Staubli VAL3: user.pjx

--- user.pjx ---
Parameters version=s7.4 stackSize=5000 millimeterUnit=true
Program file=start.pgx
Program file=stop.pgx
Data file=user.dtx

--- userPage7En.dtx ---
public num nBottomX[2]
  [0] = 21
  [1] = 21
public num nBottomY = 10
num nFirst
num nKey = 255
num nOldValue[2]
  [0] = 200
  [1] = 200
public num nPage = 100000
public num nTopX[2]
  [0] = 17
  [1] = 17
public num nTopY
public num nView
string sExample1
string sExample2
public string sItems[17]
  [0] = "Name: > "
  [1] = "coord  X > 680.52"
  [2] = "coord  Y > -61.92"
  [3] = "coord  Z > 300.32"
  [4] = "coord RX > -10   "
  [5] = "coord RY > 175.5 "
  [6] = "coord RZ > 68.47"
  [7] = "Axis pos > 90   "
  [8] = "MoveType > Linear"
  [9] = "Speed    > 600 mm/s"
  [10] = "Accelerat> 200 %"
  [11] = "Stop  > [ ]"
  [12] = "Blend[x] > 30 mm"
  [13] = "Action : 1> "
  [14] = "Action : 2> "
  [15] = "Action : 3> "
  [16] = "Anticipation > 0 mm"
string sMenu
string sMessage[3]
  [0] = "Insert the speed, all the points that"
  [1] = "have the same speeed will be change,"
  [2] = "use mm/sec >600"
string sTab[4]
  [0] = "test1"
  [1] = "test2"
  [2] = "test3"
  [3] = "test4"
string sTitle
bool Show
bool bReadWrite[17]
  [0] = true
  [1] = true
  [2] = true
  [3] = true
  [4] = true
  [5] = true
  [6] = true
  [7] = true
  [8] = true
  [9] = true
  [10] = true
  [11] = true
  [12] = true
  [13] = true
  [14] = true
  [15] = true
  [16] = true
public bool bShowDialog
public bool bUseEscape = true
public bool bUseRefresh
screen scr

--- start.pgx ---
program start()
begin
  call example1()
end

--- changeValue.pgx ---
public program changeValue(screen& x_scr, num& x_nValue[], num x_nMin, num x_nMax, num x_nX, num x_nY, string& x_sItem[])
  local num l_nOldValue[2]
  local string l_sItem
  local string l_sMessage
  local string l_sEmpty
  local bool l_bComma
begin
  //-----------------------------------------------------------------------
  //Header begin 开头
  //Description of program  程序的描述
  //  Get a numerical value on the x_nX column and x_nY line and test if    在x_nX列和x_nY行得到一个数值量，测试
  //  the value is between x_nMin and x_nMax. If the two parameters x_nMin  这个值是否在x_nMin和x_nMax之间。如果这两个参数x_nMin
  //  and x_nMax are equal there are no limits.                             和x_nMax值相等的，那这里就没有限制了。
  //  If x_sItems is not Empty, the program displays the list of Items and  如果x_sItems是非空的，程序显示了条目的列表
  //  you can change the selected Item : the index is returned in x_nValue. 你可以改变已选的条目：索引回到了x_nValue
  //
  //Input parameters  输入参数
  //  num x_nMin :    x_nMin的数值：
  //    role : min value limit  作用：最小值的限制
  //  num x_nMax :    x_nMax的数值：
  //    role : max value limit  作用：最大值的限制
  //  num x_nX :      x_nX的数值：
  //    role : X cursor position for change the value  作用：X光标的位置变化值
  //  num x_nY :      x_nY的数值
  //    role : Y cursor position for change the value  作用：Y光标的位置变化值
  //
  //Output paramaters  输出参数
  //  num x_nValue :   x_nValue的数值
  //    role : numerical value changed or index pointer of x_sItem  作用：x_sItem的数值量改变或者索引指针
  //  string x_sItems  x_sItems的字符串
  //    role : array of Items  作用：条目的数组
  //
  //Example 例子
  //  call changeValue(scrMy,l_nValue,0,10,2,5,"") //The user can changed the numerical  用户可以改变l_nValue的数值量
  //                                           value of l_nValue. If the seized          如果得到的值不在0到10范围内，
  //                                           is not between 0 to 10 the user must      用户必须改变这个值。
  //                                           changed the value.
  //
  //  call changeValue(scrMy,l_nValue,0,10,2,5,sItem) //The list sItem is displaying on  列表条目是正在显示在屏幕上，
  //                                              the screen and the user select one     用户可以选择列表中的某个元素。
  //                                              element of the list. The index         索引会回到l_nValue中。
  //                                              is returned in l_nValue.
  //
  //
  //History  历史
  //  Creation : 28-04-08 - f.Rob  创建：28-04-08 - f.Rob
  //  Modified : 08-08-11 - J.Cook 修改：08-08-11 - J.Cook
  //                                   Changed $setTextMode to setTextMode  改变$setTextMode到setTextMode
  //                                   And replaced literals ("", 0) with local variables
  //                                   when passing parameters by reference
  //
  //  Modified : 08-08-22 - J.Cook     Add screen parameter 增加屏幕参数
  //Header end  结束
  //-----------------------------------------------------------------------
  //
  if x_nMin>x_nMax
    return
  endIf
  //Print the line in white  已白色打印该行
  call nullKey(x_scr,nKey)
  l_nOldValue[1]=round(x_nValue)
  x_nValue=(round(x_nValue*100))/100
  l_nOldValue=x_nValue
  //Check if is using the comma or not  检查有没有使用逗号
  if l_nOldValue!=l_nOldValue[1]
    l_bComma=true
  else
    l_bComma=false
  endIf
  //Start  开始
  call clear(x_scr, 0,13)
  do
    if x_sItem==""
      //Use the get num  使用得到数值
      if l_bComma
        call strFill(l_sEmpty,len(toString(".2",x_nValue)),l_sEmpty)
      else
        call strFill(l_sEmpty,len(toString("",x_nValue)),l_sEmpty)
      endIf
      call type(x_scr, x_nX,x_nY,l_sEmpty)
      gotoxy(x_scr, x_nX,x_nY)
      nKey=get(x_scr, x_nValue)
      // CHECK for MIN MAX VALUE 检查最大最小值
      if x_nMax!=x_nMin
        if x_nValue>x_nMax
          //Ask if you want to continue  询问是否你想要继续
          popUpMsg("MAX: "+toString(".2",x_nMax))
          x_nValue=l_nOldValue
          //x_nValue=x_nMax
          nKey=-1
        else
          if x_nValue<x_nMin
            popUpMsg("MIN: "+toString(".2",x_nMin))
            //x_nValue=x_nMin
            x_nValue=l_nOldValue
            nKey=-1
          endIf
        endIf
      endIf
      // UPDATE THE VALUE 更新数值
      if l_bComma
        call type(x_scr, x_nX,x_nY,toString(".2",x_nValue))
      else
        call type(x_scr, x_nX,x_nY,toString("",x_nValue))
      endIf
    else
      // STRING CHOICE 字符串选择
      nKey=getKey(x_scr)
      switch nKey
        // CHANGE THE ITEMS ARRAY  改变条目数组
        case 261
          // UP
          x_nValue=abs((x_nValue+1)%size(x_sItem))
        break
        case 266
          // DOWN
          x_nValue=abs((x_nValue+size(x_sItem)-1)%size(x_sItem))
        break
      endSwitch
      // UPDATE THE VALUE 更新数值
      setTextMode(x_scr, 3)
      call typeLen(x_scr,x_nX,x_nY,x_sItem[x_nValue],10)
      setTextMode(x_scr, 0)
    endIf
    //Release the resource  释放资源
    delay(0)
  until nKey==270 or nKey==255
  if nKey==255
    bUseEscape=true
    x_nValue=l_nOldValue
    if x_sItem!=""
      x_sItem=x_sItem[l_nOldValue]
    endIf
  else
    bUseEscape=false
  endIf
  //Leave the resource  离开资源
  delay(0)
end

--- clear.pgx ---
public program clear(screen& x_scr, num x_nX, num x_nY)
  local num i
  local num lLen
begin
  //-----------------------------------------------------------------------
  //Header begin 开头
  //Description of program  程序描述
  //  Erase the pY line from the column pX of the userPage.
  //  在用户界面中，擦除pX列中的PY行
  //Input parameters  输入参数
  //  num x_nX :
  //    role : Cursor column  作用：光标列
  //    possible value : 0 to 39  可能的值：0到39
  //  num x_nY :
  //    role : Cursor row     作用：光标行
  //    possible value : 0 to 13  可能的值：0到39
  //
  //Example 例子
  //  call clear(scrMy,15,8)
  //
  //History  历史
  //  Creation : 28-04-08 - f.Rob
  //
  //  Modified : 22 Aug 2011 - J. Cook  Added user screens
  //Header end 结束
  //-----------------------------------------------------------------------
  call typeLen(x_scr, x_nX,x_nY," ",40-x_nX)
  gotoxy(x_scr, x_nX,x_nY)
end

--- divideString.pgx ---
program divideString(string& x_sMsg[], num& x_nLine[])
  local string l_sCopyMsg
  local num l_nLength
  local string l_sSwap
  local num l_nFlag
  local num l_nTotalFlag
  local string l_sCR
  local num l_nPosCR
begin
  //-----------------------------------------------------------------------
  //Header begin 开头
  //Description of program  程序描述
  //  Divide a message if it is too long.  如果它够长的话，划分一条消息
  //  The program search a space for cut the message. 程序去搜寻一个空间为的是分割消息
  //  Return the numbers of lines used for writing the message.
  //
  //Input parameters  输入参数
  //  string x_sMsg : 字符串x_sMsg
  //    role : Message that you want to display  作用：你想去展示的消息
  //  num x_sLine :   数值量x_sLine
  //    role : Numbers of the lines that will be use  作用：该行的数值将会被使用
  //
  //Example  例子
  //  call divideString("Staubli Robotics : example userPage library",l_nLine)
  //
  //History
  //  Creation : 28-04-08 - f.Rob
  //Header end 结束
  //-----------------------------------------------------------------------
  //Carriage return  回车
  l_sCR="#"
  x_nLine=0
  //Length of a line for a message 一条消息一行的长度
  l_nLength=38
  //Copy the message  复制该信息
  l_sCopyMsg=x_sMsg
  //First case  第一种情况
  call findPos(l_sCopyMsg,l_sCR,l_nPosCR)
  if (getDisplayLen(l_sCopyMsg)>l_nLength-1) or (l_nPosCR!=-1)
    //Compose the message  重组这条消息
    do
      l_sSwap=l_sCopyMsg
      //Set the x_sMsg
      if size(x_sMsg)-1<x_nLine
        insert(x_sMsg[x_nLine])
      endIf
      call findPos(l_sCopyMsg,l_sCR,l_nPosCR)
      if (getDisplayLen(l_sCopyMsg)>l_nLength-1 or (l_nPosCR!=-1)) and x_nLine<8
        //Divide the string 分割字符串
        l_nTotalFlag=0
        call findPos(l_sCopyMsg,l_sCR,l_nPosCR)
        //Divide the string
        if l_nPosCR!=-1 and l_nPosCR<l_nLength
          //Carriage return  回车
          call leftPos(l_sCopyMsg,l_nPosCR,l_sSwap)
          //l_sSwap=left(l_sCopyMsg,l_nPosCR)
          call rightPos(l_sCopyMsg,getDisplayLen(l_sCopyMsg)-(l_nPosCR)-1,l_sCopyMsg)
          //l_sCopyMsg=right(l_sCopyMsg,len(l_sCopyMsg)-(l_nPosCR)-1)
          if getDisplayLen(l_sSwap)==0
            l_sSwap=" "
          endIf
        else
          //Search for the space then return 搜索空间然后返回
          do
            call findPos(l_sSwap," ",l_nFlag)
            //l_nFlag=find(l_sSwap," ")
            if l_nFlag!=-1 and l_nFlag<=l_nLength
              //l_sSwap=right(l_sSwap,len(l_sSwap)-l_nFlag-1)
              call rightPos(l_sSwap,getDisplayLen(l_sSwap)-l_nFlag-1,l_sSwap)
              l_nTotalFlag=l_nTotalFlag+l_nFlag+1
            else
              if l_nTotalFlag==0 and (l_nFlag==-1 or l_nFlag>l_nLength)
                l_nFlag=-1
                l_nTotalFlag=38
              endIf
            endIf
          until l_nTotalFlag>=l_nLength+2 or l_nFlag==-1
          //Normal
          if l_nTotalFlag==0
            //Full line  整行
            call leftPos(l_sCopyMsg,l_nLength,l_sSwap)
            //l_sSwap=left(l_sCopyMsg,l_nLength)
            //l_sCopyMsg=right(l_sCopyMsg,len(l_sCopyMsg)-l_nLength)
            call rightPos(l_sCopyMsg,getDisplayLen(l_sCopyMsg)-l_nLength,l_sCopyMsg)
          else
            //Divide it
            call leftPos(l_sCopyMsg,l_nTotalFlag-l_nFlag-2,l_sSwap)
            //l_sSwap=left(l_sCopyMsg,l_nTotalFlag-l_nFlag-2)
            //l_sCopyMsg=right(l_sCopyMsg,len(l_sCopyMsg)-(l_nTotalFlag-l_nFlag-1))
            call rightPos(l_sCopyMsg,getDisplayLen(l_sCopyMsg)-(l_nTotalFlag-l_nFlag-1),l_sCopyMsg)
          endIf
        endIf
        //Set the string  设置字符串
        x_sMsg[x_nLine]=l_sSwap
        x_nLine=x_nLine+1
      else
        //Limit the string  限制字符串
        call rightPos(l_sSwap,l_nLength,x_sMsg[x_nLine])
        //x_sMsg[x_nLine]=right(l_sSwap,l_nLength)
        l_sSwap=""
      endIf
    until l_sSwap==""
  endIf
end

--- editNumField.pgx ---
public program editNumField(screen& x_scr, string x_sTitle, string& x_sItemName[], num& x_nItem[], num& x_nMin[], num& x_nMax[])
  local num j
  local num l_nSize
  local num l_nKey
  local string l_sEvent
  local num l_nIndex
  local num l_nField
  local string l_sItem
  local string l_sEmpty
begin
  //-----------------------------------------------------------------------
  //Header begin 开头
  //Description of program  程序描述
  //  Modify numerical values of a list of Items. 修改条目列表的数值量
  //  When you use this program it creates automatically the list of x_sItemName. 当你使用这个程序，它能够自动创建x_sItemName的列表
  //  You can navigate and select the Item that you want to modify the value.     你能够导航和选择你想修改值的条目
  //  If you press on ESC you quit this list and all values that you have entered 如果你按压ESC键，你会退出这个列表，你已经输入的所有值
  //  will not be saved.                                                          将不会被保存
  //  You can use an array for the parameters min and max to add limits           你能够使用一个针对最小值最大值的参数的数组去增加
  //  for every Items.                                                            每一个条目的限制
  //  If the parameters min and max are equal there are no limits.                如果参数的最小值和最大值是相等的，那儿就没有限制。
  //
  //Input parameters  输入参数：
  //  string x_sTitle :  字符串x_sTitle
  //    role : Title of the list  作用：列表的标题
  //
  //Output parameters  输出参数
  //  string x_sItemName : 字符串x_sItemName：
  //    role : array of Items that you want to edit the numerical values 作用：你想要编辑的条目数组的数值量
  //  num x_nItem :  数值量x_nItem
  //    role : array of values corresponding of the Items  作用：对应条目的数组值
  //  num x_nMin :  数值量x_nMin
  //    role : minimum limit for x_nItem values  作用：x_nItem值的最小值限制
  //  num x_nMax    数值量x_nMax
  //    role : maximum limit for x_nItem values  作用：x_nItem值的最大值限制
  //
  //Example 例子
  //  call editNumField(scrMy,"Menu",sItem,nItem,nMin,nMax)
  //
  //History
  //  Creation : 28-04-08 - f.Rob
  //  Modified : 08-08-11 - J.Cook     Changed $setTextMode to setTextMode
  //                                   And replaced literals ("", 0) with local variables
  //                                   when passing parameters by reference
  //
  //  Modified : 08-08-22 - J.Cook     Add screen parameter
  //Header end 结束
  //-----------------------------------------------------------------------
  l_sEmpty = ""
  nView=nFirst=0
  //Copy all the values x_nItem 复制所有的x_nItem的值
  call numCopy(x_nItem,nOldValue)
  l_nSize=size(x_nItem)-1
  //Create the LIST  创建列表
  call setSizeList(7,max((6-l_nSize/2)-2,2),23,min((l_nSize+1),8))
  call listCreate(x_scr, x_sTitle)
  //Insert Items  插入条目
  for j=0 to l_nSize
    l_sItem=x_sItemName[j]
    call strlength(l_sItem,15)
    call listAdd(l_sItem+": "+toString(".1",x_nItem[j]))
  endFor
  call listUpdate(x_scr, 0)
  do
    call clear(x_scr, 0,13)
    call typeMenu(x_scr, 8,"OK")
    l_nKey=get(x_scr)
    call listEvent(x_scr, l_nKey,l_nIndex,l_sEvent)
    //On Enter Key  在回车键
    if l_nKey==270
      call listCursor(x_scr,nView,false)
      if size(x_nMin)==size(x_nItem)
        //Use min and max  使用最小值和最大值
        call changeValue(x_scr, x_nItem[l_nIndex],x_nMin[l_nIndex],x_nMax[l_nIndex],15+10,nView+nTopY+1,l_sEmpty)
      else
        call changeValue(x_scr,x_nItem[l_nIndex],0,0,15+10,nView+nTopY+1,l_sEmpty)
      endIf
      //UPDATE 更新
      call listDel(l_nIndex)
      l_sItem=x_sItemName[l_nIndex]
      call strlength(l_sItem,15)
      call listIns(l_sItem+": "+toString(".1",x_nItem[l_nIndex]),l_nIndex)
      call listUpdate(x_scr,l_nIndex-nView)
    endIf
    delay(0)
  until l_nKey==278 or l_nKey==255
  //Escape use????
  if l_nKey==255
    bUseEscape=true
    call numCopy(nOldValue,x_nItem)
  else
    bUseEscape=false
  endIf
  //Exit
  call nullKey(x_scr,l_nKey)
end

--- example.pgx ---
program example()
  local num l_nKey
  local num l_nItem[2]
  local num l_nView[2]
  local string l_sItem
  local string l_sMsg
  local string l_sButton[2]
  local num i
  local bool l_bLarge
  local bool l_bQuit
  local string l_sMenu
  local num l_nSeconds
  local string l_sHourMinSec
  local string l_sItemName[5]
  local num l_nItemExample[5]
  local num l_nMaxExample[5]
  local num l_nMinExample[5]
  local num l_nMenu
  local num l_nSelected[2]
  local bool l_bExit
  local num l_nFirst[2]
  local string l_sEmpty
  local string l_sText
  local num l_nZero
begin
  //-----------------------------------------------------------------------
  //Header begin 开头
  //Description of program 程序的描述
  //  This is an example for use this library. 这是一个使用库的例子程序。
  //  This example performs the following actions : 该程序执行以下动作：
  //  - Run the fhmns program (converted of num seconds in string hour) 运行fhmns程序(时间转换程序，把秒数转换成几时几分几秒的形式)
  //  - add, insert, delete, and select an Item with an updating of the menu. 用一个更新的菜单显示增加，插入，删除和选择一个条目
  //  - change Menu (list of Items) with left and right keys 用左右键改变菜单（条目列表）
  //  - clear the menu  清除菜单
  //  - Run a simple list (no array) for just test the scrolling 运行一个简单的列表（没有数组），只为了测试列表滚动条
  //
  //  The sequence is : 这个顺序是：
  //  - Creation of 2 string arrays for the lists of items 条目列表里创建两个字符串数组
  //  - Start main loop 开始主循环
  //  -   Creation of the menu with 2 lists  2个列表菜单的创建
  //  -   Reading events from the keyboard   从键盘中读取事件
  //  -     case TAB           : update the width of the list (enlarge/reduce)  TAB键：更新列表的宽度（扩大/减少）
  //  -     case left or right : update the item's list and change the menu    左右键：更新条目的列表和改变菜单
  //  -     case Enter         : displays the Item selected                    回车键：显示已选的条目
  //  -     case F1 or ESC     : quit the program                           F1或ESC键：退出程序
  //  -     case F2            : clear th list                                   F2键：清除列表
  //  -     case F3            : Run function wich converted seconds             F3键：运行时间转换函数
  //                              -> string Hours:Min:Sec                              由s转换成h：m：s的形式
  //  -     case F4            : test editNumField() function                    F4键：测试editNumField()函数
  //  -     case F5            : creation of an other list : simple list         F5键：创建一个其他列表：简单列表
  //  -     case F6            : delete an Item                                  F6键：删除一个条目
  //  -     case F7            : add an item at the end of the list              F7键：在列表末端增加一个条目
  //  -     case F8            : insert an item at the current position          F8键：在当前的位置插入一个条目
  //  -   Update the Item's list                                                 更新条目的列表
  //  -   Refresh the screen                                                     刷新屏幕
  //
  //History                                                                      历史
  //  Creation : 28-04-08 - f.Rob                                                创建：28-04-08 - f.Rob
  //  Modified : 08-08-11 - J.Cook     Changed $setTextMode to setTextMode       修改：08-08-11 - J.Cook
  //                                   And replaced literals ("", 0) with local variables
  //                                   when passing parameters by reference
  //Header end  结束
  //-----------------------------------------------------------------------
  l_sEmpty = ""
  cls(scr)
  userPage(scr)
  //---------------------------------------------------
  // CREATION OF 2 STRING ARRAYS FOR THE LISTS OF ITEMS 为这个项目的列表创建2字符串数组
  //---------------------------------------------------
  //Empty the two lists  清空这两个列表
  call stringCopy(l_sEmpty,sExample1)
  call stringCopy(l_sEmpty,sExample2)
  //Build the first list  建立第一个列表
  for i=0 to 19
    if sExample1!=""
      append(sExample1)
    endIf
    sExample1[i]="Program "+toString("",i)
  endFor
  //Build the second list  建立第二个列表
  for i=0 to 14
    if sExample2!=""
      append(sExample2)
    endIf
    sExample2[i]="Item "+toString("",i)
  endFor
  //----------------
  // START THE LOOP   开始循环
  //----------------
  do
    //-------------------------------------
    // CREATION OF THE MENU WITH TWO LISTS   创建带两个列表的菜单
    //-------------------------------------
    title(scr,"userPage example")
    //Creation size of the list    创建列表的大小
    call setSizeList(20,0,18,11)
    //Enlarge/reduce the width of the list menu when tab is pressed  扩大/减小列表惨淡的宽度，当按tab键
    call setView(l_bLarge)
    //Refresh the list     刷新列表
    call listCreate(scr,"Menu "+toString("",l_nMenu+1))
    switch l_nMenu
      //Insert all the array into the list  插入所有的数组进入列表
      case 0
        call listAdd(sExample1)
      break
      case 1
        call listAdd(sExample2)
      break
    endSwitch
    //Refresh cursor position - selected item  刷新光标位置-选择条目
    call selectNewField(scr,l_nSelected[l_nMenu],l_nItem[l_nMenu],l_nView[l_nMenu])
    //Menu  菜单
    l_sMenu="Exit,Clean,Conversion,Parameter,Simple list,Delete,Add,Insert"
    call stringToArray(l_sMenu,sMenu)
    if !l_bLarge
      //Set the menu at the Y position : 3  设置菜单在Y方向上为3
      call setMenu(scr,sMenu,true,3)
    else
      //Displays the menu on the bottom side not on the left side  显示菜单在底部滑动条上而不是在左边的滑动条上
      call setMenu(scr,sMenu,true,-1)
    endIf
    //-----------------------------------
    //  READING EVENTS FROM THE KEYBOARD   从键盘中读取事件
    //-----------------------------------
    l_nKey=get(scr)
    call listEvent(scr,l_nKey,l_nItem[l_nMenu],l_sItem)
    //Update the cursor position viewing on the screen  更新屏幕上显示的光标位置
    //The two lists are independent so utilisation of an array with two elements  这两个列表是独立的，利用的是两个元素的一个数组
    l_nView[l_nMenu]=nView
    //Update the selection of the Item  更新条目的选择
    l_nSelected[l_nMenu]=l_nItem[l_nMenu]
    switch (l_nKey)
      //Tab  Tab键
      //------------------------------------------------
      //  UPDATE THE WIDTH OF THE LIST (ENLARGE/REDUCE)   更新列表的宽度（扩大/缩小）
      //------------------------------------------------
      case 259
        //Variable corresponding to Enlarge/Reduce the width of the list  变量对应的是扩大/缩小列表的宽度
        l_bLarge=!l_bLarge
      break
      //Left or Right 左边或右边
      //---------------------------------------------
      //  UPDATE THE ITEM'S LIST AND CHANGE THE MENU  更新条目的列表和改变菜单
      //---------------------------------------------
      case 264,268
        switch l_nMenu
          case 0
            call stringCopy(sItems,sExample1)
          break
          case 1
            call stringCopy(sItems,sExample2)
          break
        endSwitch
        //Update l_nMenu  更新l_nMenu
        if l_nKey==264
          //Right   右边
          //Increment l_nMenu   l_nMenu的增加
          l_nMenu=abs(l_nMenu-1)%2
        else
          //Left    左边
          //Decrement l_nMenu   l_nMenu的减少
          l_nMenu=abs(l_nMenu+1)%2
        endIf
        //Update the selected item  更新已选的条目
        l_nSelected[l_nMenu]=l_nItem[l_nMenu]
      break
      //Enter   回车
      //-----------------------------
      //  DISPLAYS THE ITEM SELECTED  显示已选的条目
      //-----------------------------
      case 270
        //No action just displays a message, it's an example  没有动作仅仅显示一条信息，这是一个列子
        call timerDialog(scr,"Selected item: "+l_sItem,1)
      break
      //F1  F1键
      //-------------------
      //  QUIT THE PROGRAM   退出程序
      //-------------------
      case 271
        //Creation of two buttons functions  创建两个按键函数
        //l_sButton    : F8  l_sButton：F8键
        //l_sButton[1] : F7  l_sButton[1]：F7键
        l_sButton="Yes"
        l_sButton[1]="No"
        call questionDialog(scr,"Do you want to quit ?",l_sButton,l_nKey)
        //"Enter" or "F8" pressed   按"回车"或者按"F8"
        if l_nKey==0 or l_nKey==1
          l_bQuit=true
        endIf
        cls(scr)
      break
      //F2  F2键
      //-----------------
      //  CLEAR THE LIST  清除列表
      //-----------------
      case 272
        //Creation of two buttons functions  创建两个按键函数
        //l_sButton    : F8  l_sButton：F8键
        //l_sButton[1] : F7  l_sButton[1]：F7键
        l_sButton="Yes"
        l_sButton[1]="No"
        call questionDialog(scr,"Do you want to clear the list ?",l_sButton,i)
        if i==0 or i==1
          call listEmpty()
        endIf
      break
      //F3  F3键
      //--------------------------------------------------------------
      //  RUN FUNCTION WICH CONVERTED SECONDS -> STRING HOURS:MIN:SEC  运行时间转换函数：把秒数转换成几时几分几秒的形式
      //--------------------------------------------------------------
      case 273
        cls()
        call insertDialog(scr,"Number of seconds that you want to convert in Hour:min:sec : #",l_nSeconds,0,0)
        call fhmns(l_nSeconds,l_sHourMinSec)
        popUpMsg("Conversion : "+l_sHourMinSec)
      break
      //F4  F4键
      //---------------------------------
      //  TEST " EDITNUMFIELD " FUNCTION  测试 "EDITNUMFIELD" 函数
      //---------------------------------
      case 274
        //Test editNumField function   测试editNumField函数
        for i=0 to size(l_sItemName)-1
          l_sItemName[i]="Item "+toString("",i)
          //No Limits for all  对所有的情况都没有限制
          l_nMinExample[i]=0
          l_nMaxExample[i]=0
        endFor
        call editNumField(scr,"Change Parameter",l_sItemName,l_nItemExample,l_nMinExample,l_nMaxExample)
      break
      // F5  F5键
      //------------------------------------------
      //  CREATION OF AN OTHER LIST : SIMPLE LIST  一个其他列表的创建：简单列表
      //------------------------------------------
      case 275
        //Simple list for test the scrolling 简单列表为了来测试滚动条
        cls(scr)
        do
          l_bExit=false
          //Size of the list 列表的大小
          call setSizeList(20,0,18,11)
          //Creation of the list with the title "Simple list"  创建一个题为"Simple list"列表
          call listCreate(scr,"Simple list")
          //Add Items in the list  在列表中增加条目
          l_sText = "Item 1"
          call listAdd(l_sText)
          l_sText = "Item 2"
          call listAdd(l_sText)
          l_sText = "Item 3"
          call listAdd(l_sText)
          l_sText = "Item 4"
          call listAdd(l_sText)
          //Update the list  更新列表
          call listUpdate(scr,0)
          call typeMenu(scr,1,"Quit simple list")
          i=get(scr)
          l_nZero = 0
          call listEvent(scr,i,l_nZero,l_sEmpty)
          switch i
            case 271,255
              l_sButton="Yes"
              l_sButton[1]="No"
              call questionDialog(scr,"Do you want to quit this program ?",l_sButton,i)
              //"Enter" or "F8" pressed  按回车键或者F8键
              if i==0 or i==1
                l_bExit=true
              else
                cls(scr)
              endIf
            break
          endSwitch
        until l_bExit
      break
      //F6  F6键
      //-----------------
      //  DELETE AN ITEM  删除一个条目
      //-----------------
      case 276
        //Delete  删除
        l_sButton="Yes"
        l_sButton[1]="No"
        call questionDialog(scr,"Do you want to delete "+l_sItem+" ?",l_sButton,i)
        if i==0 or i==1
          call listDel(l_nItem[l_nMenu])
        endIf
      break
      //F7  F7键
      //---------------------------------
      //  ADD AN ITEM AT END OF THE LIST  在末尾增加列表的一个条目
      //---------------------------------
      case 277
        call timerDialog(scr,"Add One element #",0)
        l_sItem="new Item"
        //Read one string from the keyboard and write it on the  从键盘上读取一个字符串和把它写入到第15列第7行
        //15 column and 7 line.
        call read(scr,15,7,l_sItem,10,false)
        if !bUseEscape
          call listAdd(l_sItem)
        endIf
        switch l_nMenu
          case 0
            l_nSelected=size(sExample1)
          break
          case 1
            l_nSelected=size(sExample2)
          break
        endSwitch
      break
      //F8  F8键
      //-----------------------------------------
      //  INSERT AN ITEM AT THE CURRENT POSITION  在当前位置插入一个条目
      //-----------------------------------------
      case 278
        //Insert at the current position  在当前位置插入
        call timerDialog(scr,"Insert One element #",0)
        l_sItem="new Item"
        call read(scr,15,7,l_sItem,10,false)
        if !isKeyPressed(255) and l_sItem!="new Item"
          call listIns(l_sItem,l_nItem[l_nMenu])
        endIf
      break
    endSwitch
    //-------------------------
    //  UPDATE THE ITEM'S LIST  更新条目列表
    //-------------------------
    //Update the list  更新列表
    switch l_nKey
      case 272,276,277,278
        //Update the item's list with the global variable 用全局变量来更新条目的列表
        switch l_nMenu
          case 0
            call stringCopy(sItems,sExample1)
          break
          case 1
            call stringCopy(sItems,sExample2)
          break
        endSwitch
      break
    endSwitch
    //-------------------
    //REFRESH THE SCREEN  刷新屏幕
    //-------------------
    if l_nKey>=270 and l_nKey<=278 or l_nKey==259
      cls(scr)
    endIf
    delay(0)
  until l_bQuit
end

--- example1.pgx ---
program example1()
  local num l_nKey
  local num l_nItem[2]
  local num l_nView[2]
  local string l_sItem
  local string l_sMsg
  local string l_sButton[2]
  local num i
  local bool l_bLarge
  local bool l_bQuit
  local string l_sMenu
  local num l_nSeconds
  local string l_sHourMinSec
  local string l_sItemName[5]
  local num l_nItemExample[5]
  local num l_nMaxExample[5]
  local num l_nMinExample[5]
  local num l_nMenu
  local num l_nSelected[2]
  local bool l_bExit
  local num l_nFirst[2]
  local string l_sEmpty
  local string l_sText
  local num l_nZero
begin
  //-----------------------------------------------------------------------
  //Header begin 开头
  //Description of program 程序的描述
  //  This is an example for use this library. 这是一个使用库的例子程序。
  //  This example performs the following actions : 该程序执行以下动作：
  //  - Run the fhmns program (converted of num seconds in string hour) 运行fhmns程序(时间转换程序，把秒数转换成几时几分几秒的形式)
  //  - add, insert, delete, and select an Item with an updating of the menu. 用一个更新的菜单显示增加，插入，删除和选择一个条目
  //  - change Menu (list of Items) with left and right keys 用左右键改变菜单（条目列表）
  //  - clear the menu  清除菜单
  //
  //
  //  The sequence is : 这个顺序是：
  //  - Creation of 2 string arrays for the lists of items 条目列表里创建两个字符串数组
  //  - Start main loop 开始主循环
  //  -   Creation of the menu with 2 lists  2个列表菜单的创建
  //  -   Reading events from the keyboard   从键盘中读取事件
  //  -     case TAB           : update the width of the list (enlarge/reduce)  TAB键：更新列表的宽度（扩大/减少）
  //  -     case left or right : update the item's list and change the menu    左右键：更新条目的列表和改变菜单
  //  -     case Enter         : displays the Item selected                    回车键：显示已选的条目
  //  -     case F1 or ESC     : quit the program                           F1或ESC键：退出程序
  //  -     case F2            : clear th list                                   F2键：清除列表
  //  -     case F3            : Run function wich converted seconds             F3键：运行时间转换函数
  //                              -> string Hours:Min:Sec                              由s转换成h：m：s的形式
  //  -     case F4            : test editNumField() function                    F4键：测试editNumField()函数
  //  -     case F5            : delete an Item                                  F5键：删除一个条目
  //  -     case F6            : insert an item at the current position          F6键：在当前的位置插入一个条目
  //  -   Update the Item's list                                                 更新条目的列表
  //  -   Refresh the screen                                                     刷新屏幕
  //
  //History                                                                      历史
  //  Creation : 28-04-08 - f.Rob                                                创建：28-04-08 - f.Rob
  //  Modified : 08-08-11 - J.Cook     Changed $setTextMode to setTextMode       修改：08-08-11 - J.Cook
  //                                   And replaced literals ("", 0) with local variables
  //                                   when passing parameters by reference
  //Header end  结束
  //-----------------------------------------------------------------------
  l_sEmpty = ""
  cls(scr)
  userPage(scr)
  //---------------------------------------------------
  // CREATION OF 2 STRING ARRAYS FOR THE LISTS OF ITEMS 为这个项目的列表创建2字符串数组
  //---------------------------------------------------
  //Empty the two lists  清空这两个列表
  call stringCopy(l_sEmpty,sExample1)
  call stringCopy(l_sEmpty,sExample2)
  //Build the first list  建立第一个列表
  for i=0 to 19
    if sExample1!=""
      append(sExample1)
    endIf
    sExample1[i]="Program "+toString("",i)
  endFor
  //Build the second list  建立第二个列表
  for i=0 to 14
    if sExample2!=""
      append(sExample2)
    endIf
    sExample2[i]="Item "+toString("",i)
  endFor
  //----------------
  // START THE LOOP   开始循环
  //----------------
  do
    //-------------------------------------
    // CREATION OF THE MENU WITH TWO LISTS   创建带两个列表的菜单
    //-------------------------------------
    title(scr,"userPage example")
    //Creation size of the list    创建列表的大小
    call setSizeList(20,0,18,11)
    //Enlarge/reduce the width of the list menu when tab is pressed  扩大/减小列表惨淡的宽度，当按tab键
    call setView(l_bLarge)
    //Refresh the list     刷新列表
    call listCreate(scr,"Menu "+toString("",l_nMenu+1))
    switch l_nMenu
      //Insert all the array into the list  插入所有的数组进入列表
      case 0
        call listAdd(sExample1)
      break
      case 1
        call listAdd(sExample2)
      break
    endSwitch
    //Refresh cursor position - selected item  刷新光标位置-选择条目
    call selectNewField(scr,l_nSelected[l_nMenu],l_nItem[l_nMenu],l_nView[l_nMenu])
    //Menu  菜单
    l_sMenu="Exit,Clean,Conversion,Parameter,Delete,Insert"
    call stringToArray(l_sMenu,sMenu)
    if !l_bLarge
      //Set the menu at the Y position : 3  设置菜单在Y方向上为3
      call setMenu(scr,sMenu,true,3)
    else
      //Displays the menu on the bottom side not on the left side  显示菜单在底部滑动条上而不是在左边的滑动条上
      call setMenu(scr,sMenu,true,-1)
    endIf
    //-----------------------------------
    //  READING EVENTS FROM THE KEYBOARD   从键盘中读取事件
    //-----------------------------------
    l_nKey=get(scr)
    call listEvent(scr,l_nKey,l_nItem[l_nMenu],l_sItem)
    //Update the cursor position viewing on the screen  更新屏幕上显示的光标位置
    //The two lists are independent so utilisation of an array with two elements  这两个列表是独立的，利用的是两个元素的一个数组
    l_nView[l_nMenu]=nView
    //Update the selection of the Item  更新条目的选择
    l_nSelected[l_nMenu]=l_nItem[l_nMenu]
    switch (l_nKey)
      //Tab  Tab键
      //------------------------------------------------
      //  UPDATE THE WIDTH OF THE LIST (ENLARGE/REDUCE)   更新列表的宽度（扩大/缩小）
      //------------------------------------------------
      case 259
        //Variable corresponding to Enlarge/Reduce the width of the list  变量对应的是扩大/缩小列表的宽度
        l_bLarge=!l_bLarge
      break
      //Left or Right 左边或右边
      //---------------------------------------------
      //  UPDATE THE ITEM'S LIST AND CHANGE THE MENU  更新条目的列表和改变菜单
      //---------------------------------------------
      case 264,268
        switch l_nMenu
          case 0
            call stringCopy(sItems,sExample1)
          break
          case 1
            call stringCopy(sItems,sExample2)
          break
        endSwitch
        //Update l_nMenu  更新l_nMenu
        if l_nKey==264
          //Right   右边
          //Increment l_nMenu   l_nMenu的增加
          l_nMenu=abs(l_nMenu-1)%2
        else
          //Left    左边
          //Decrement l_nMenu   l_nMenu的减少
          l_nMenu=abs(l_nMenu+1)%2
        endIf
        //Update the selected item  更新已选的条目
        l_nSelected[l_nMenu]=l_nItem[l_nMenu]
      break
      //Enter   回车
      //-----------------------------
      //  DISPLAYS THE ITEM SELECTED  显示已选的条目
      //-----------------------------
      case 270
        //No action just displays a message, it's an example  没有动作仅仅显示一条信息，这是一个列子
        call timerDialog(scr,"Selected item: "+l_sItem,1)
      break
      //F1  F1键
      //-------------------
      //  QUIT THE PROGRAM   退出程序
      //-------------------
      case 271
        //Creation of two buttons functions  创建两个按键函数
        //l_sButton    : F8  l_sButton：F8键
        //l_sButton[1] : F7  l_sButton[1]：F7键
        l_sButton="Yes"
        l_sButton[1]="No"
        call questionDialog(scr,"Do you want to quit ?",l_sButton,l_nKey)
        //"Enter" or "F8" pressed   按"回车"或者按"F8"
        cls(scr)
        if l_nKey==0 or l_nKey==1
          l_bQuit=true
        endIf
      break
      //F2  F2键
      //-----------------
      //  CLEAR THE LIST  清除列表
      //-----------------
      case 272
        //Creation of two buttons functions  创建两个按键函数
        //l_sButton    : F8  l_sButton：F8键
        //l_sButton[1] : F7  l_sButton[1]：F7键
        l_sButton="Yes"
        l_sButton[1]="No"
        call questionDialog(scr,"Do you want to clear the list ?",l_sButton,i)
        if i==0 or i==1
          call listEmpty()
        endIf
      break
      //F3  F3键
      //--------------------------------------------------------------
      //  RUN FUNCTION WICH CONVERTED SECONDS -> STRING HOURS:MIN:SEC  运行时间转换函数：把秒数转换成几时几分几秒的形式
      //--------------------------------------------------------------
      case 273
        cls()
        call insertDialog(scr,"Number of seconds that you want to convert in Hour:min:sec : #",l_nSeconds,0,0)
        call fhmns(l_nSeconds,l_sHourMinSec)
        popUpMsg("Conversion : "+l_sHourMinSec)
      break
      //F4  F4键
      //---------------------------------
      //  TEST " EDITNUMFIELD " FUNCTION  测试 "EDITNUMFIELD" 函数
      //---------------------------------
      case 274
        //Test editNumField function   测试editNumField函数
        for i=0 to size(l_sItemName)-1
          l_sItemName[i]="Item "+toString("",i)
          //No Limits for all  对所有的情况都没有限制
          l_nMinExample[i]=0
          l_nMaxExample[i]=0
        endFor
        call editNumField(scr,"Change Parameter",l_sItemName,l_nItemExample,l_nMinExample,l_nMaxExample)
      break

      //F5  F5键
      //-----------------
      //  DELETE AN ITEM  删除一个条目
      //-----------------
      case 275
        //Delete  删除
        l_sButton="Yes"
        l_sButton[1]="No"
        call questionDialog(scr,"Do you want to delete "+l_sItem+" ?",l_sButton,i)
        if i==0 or i==1
          call listDel(l_nItem[l_nMenu])
        endIf
      break

      //F6  F6键
      //-----------------------------------------
      //  INSERT AN ITEM AT THE CURRENT POSITION  在当前位置插入一个条目
      //-----------------------------------------
      case 276
        //Insert at the current position  在当前位置插入
        call timerDialog(scr,"Insert One element #",0)
        l_sItem="new Item"
        call read(scr,15,7,l_sItem,10,false)
        if !isKeyPressed(255) and l_sItem!="new Item"
          call listIns(l_sItem,l_nItem[l_nMenu])
        endIf
      break
    endSwitch
    //-------------------------
    //  UPDATE THE ITEM'S LIST  更新条目列表
    //-------------------------
    //Update the list  更新列表
    switch l_nKey
      case 272,275,276
        //Update the item's list with the global variable 用全局变量来更新条目的列表
        switch l_nMenu
          case 0
            call stringCopy(sItems,sExample1)
          break
          case 1
            call stringCopy(sItems,sExample2)
          break
        endSwitch
      break
    endSwitch
    //-------------------
    //REFRESH THE SCREEN  刷新屏幕
    //-------------------
    if l_nKey>=270 and l_nKey<=276 or l_nKey==259
      cls(scr)
    endIf
    delay(0)
  until l_bQuit
end

--- fhmns.pgx ---
public program fhmns(num x_nSec, string& x_sHMinSec[])
  local num l_nHour
  local num l_nMin
  local num l_nSec
begin
  //-----------------------------------------------------------------------
  //Header begin 开头
  //Description of program  程序描述
  //  Convert a num seconds in string hour : "xx h xx mn xx s".
  //  把时间的秒数转变成"xx h xx mn xx s"的形式
  //Input parameters  输入参数
  //  num x_nSec : 数值量x_nSec
  //    role : put a numerical expression that you want to convert in Hmns
  //    作用：放一个数值的表达式，这个表达式是你想去转换的
  //Output parameters  输出参数
  //  string x_sHMinSec :  字符串x_sHMinSec
  //    role : string hour correspond of your numerical expression
  //    作用：对应于你的数值表达式的字符串小时
  //Example
  //  call hmns(l_nSecond,l_sHMinSec)
  //
  //History
  //  Creation : 28-04-08 - f.Rob
  //Header end
  //-----------------------------------------------------------------------
  l_nHour=roundDown(x_nSec/3600)
  l_nMin=roundDown((x_nSec%3600)/60)
  l_nSec=roundDown(x_nSec-l_nHour*3600-l_nMin*60)
  x_sHMinSec=toString("3.0",l_nHour)+" h "+toString("2.0",l_nMin)+" mn "+toString("2.0",l_nSec)+" s"
end

--- findPos.pgx ---
public program findPos(string x_sText1, string x_sText2, num& x_nPos[])
  local num l_nPos
begin
  //-----------------------------------------------------------------------
  //Header begin  开头
  //Description of program  程序描述
  //  This program is identical "find()" but it accepts Chinese characters 这个程序是与"find()"是相同的，但是它还能接受中文字符
  //  Returns the index of the first character in the first occurrence  在sText1的sText2第一次出现的地方返回第一个字符的索引
  //  of sText2 in sText1.
  //  If sText2 does not appear in sText1, the instruction returns -1.  如果sText2没有出现在sText1中，该指令返回-1
  //
  //
  //Input parameters  输入参数
  //  string x_sItem1 and x_sItem2 : 字符串x_sItem1和x_sItem2
  //    role : string 1 to compare with the string 2  作用：字符串2和字符串1相比较
  //  num x_nPos : 数值 x_nPos
  //    role : index of the first character in the first occurrence  作用：在sText1的sText2第一次出现的地方返回第一个字符的索引
  //  of sText2 in sText1
  //
  //Example  例子
  //  call findPos()
  //
  //History
  //  Creation : 28-04-08 - f.Rob
  //Header end  结束
  //-----------------------------------------------------------------------
  // Find the char using getDisplayLen 找到使用getDisplayLen的字符
  l_nPos=find(x_sText1,x_sText2)
  if l_nPos!=-1
    x_nPos=getDisplayLen(left(x_sText1,l_nPos))
  else
    x_nPos=-1
  endIf
end

--- getListPosition.pgx ---
public program getListPosition(num& x_nIndexX[], num& x_nIndexY[])
begin
  //-----------------------------------------------------------------------
  //Header begin 开头
  //Description of program  程序描述
  //  Returns the position of the list menu. 返回列表菜单的位置。
  //
  //Input parameters  输入参数
  //  num x_nIndexX : 数值x_nIndexX
  //    role : cursor column position : top left corner for the beginning of the list menu
  //    作用：光标列的位置：左上角开始菜单列表
  //  num x_nIndexY : 数值x_nIndexY
  //    role : cursor column position : top left corner for the beginning of the list menu
  //    作用：光标列的位置：左上角开始菜单列表
  //History
  //  Creation : 28-04-08 - f.Rob
  //Header end
  //-----------------------------------------------------------------------
  x_nIndexX=nTopX+1
  x_nIndexY=nFirst+nView+nTopY+1
end

--- getMenu.pgx ---
public program getMenu(string& x_sMenu[], bool& x_bUseMenu[])
  local num i
begin
  //-----------------------------------------------------------------------
  //Header begin 开头
  //Description of program  程序描述
  //  Returns the status of all the elements of the x_sMenu array.  返回x_sMenu数组所有元素的状态
  //  If an element is empty, the program returns "true" for the   如果一个元素示空值，程序返回"真"对于
  //  corresponding element in x_bUseMenu[ ].                      相对应的在x_bUseMenu[ ]的元素。
  //
  //Output parameters  输出参数
  //  string x_sMenu :  字符串x_sMenu
  //    role : It's an array of string, every elements represent an Item for the
  //    作用: 这是一个字符串数组，每个元素代表菜单的一个条目。
  //    menu.
  //  bool x_bUseMenu : 布尔量x_bUseMenu
  //    role : Status of all the Element of the x_sMenu array.
  //    作用：x_sMenu数组的所有元素状态
  //Example
  //  call getMenu(sMenu,l_bUseMenu)
  //
  //History
  //  Creation : 28-04-08 - f.Rob
  //Header end
  //-----------------------------------------------------------------------
  for i=0 to (size(x_bUseMenu)-1)
    x_bUseMenu[i]=false
    if (size(x_sMenu)-1)>=i
      //Element not empty
      if x_sMenu[i]!=""
        //Active the button
        x_bUseMenu[i]=true
      endIf
    endIf
  endFor
end

--- getView.pgx ---
public program getView(bool& x_bView[])
begin
  //-----------------------------------------------------------------------
  //Header begin
  //Description of program
  //  This program returns true in x_bView if the menu of the list
  //  is displayed in full-page and false otherwise.
  //  这个程序当整个菜单列表全屏显示的时候，返回在x_bView的真值，否则为假。
  //Output parameters  输出参数
  //  bool x_bView : 布尔量x_bView
  //    role : Status of the size of list menu.
  //    作用：菜单列表的大小状态
  //    possible values : true when the list menu is displayed in full-page,
  //                      false otherwise.
  //    可能的值：当菜单列表全屏显示时，返回真值，否则为假。
  //Example
  //  call getView(l_bView)
  //
  //History
  //  Creation : 28-04-08 - f.Rob
  //Header end
  //-----------------------------------------------------------------------
  if nBottomX==38
    x_bView=true
  else
    x_bView=false
  endIf
end

--- hmns.pgx ---
public program hmns(num x_nSec, num& x_nHour[], num& x_nMinute[], num& x_nSecond[])
begin
  //-----------------------------------------------------------------------
  //Header begin
  //Description of program
  //  Decompose num seconds in num Hours,minutes, seconds.
  //  分解数值量的秒数为几时几分几秒的形式
  //Input parameters  输入参数
  //  num x_nSec : 数值量x_nSec
  //    role : put a numerical expression that you want to convert in Hmns
  //    作用：放一个你想转换成Hmns形式的秒数数值表达式
  //Output parameters 输出参数
  //  num x_nHour : 数值量x_nHour
  //    role : numerical expression that contains Hours
  //    作用：包含小时的数值量表达式
  //  num x_nMinute :数值量x_nMinute
  //    role : numerical expression that contains Minutes
  //    作用：包含分钟的数值量表达式
  //  num x_nSecond :数值量x_nSecond
  //    role : numerical expression that contains Seconds
  //    作用：包含秒数的数值量表达式
  //Example
  //  call hmns(54200,l_nHour,l_nMinute,l_nSecond)
  //
  //History
  //  Creation : 28-04-08 - f.Rob
  //Header end
  //-----------------------------------------------------------------------
  x_nHour=roundDown(x_nSec/3600)
  x_nMinute=roundDown((x_nSec%3600)/60)
  x_nSecond=roundDown(x_nSec-x_nHour*3600-x_nMinute*60)
end

--- insertDialog.pgx ---
public program insertDialog(screen& x_scr, string x_sMsg, num& x_nItem[], num x_nMin, num x_nMax)
  local num l_nStartLine
  local num l_nLine
  local num i
  local num l_nPX
  local num l_nPY
  local string l_sItem
  local string l_sMessage
  local string l_sEmpty
begin
  //-----------------------------------------------------------------------
  //Header begin
  //Description of program
  //  Modify the x_sItem, using a min max range. 修改x_sItem，使用一个最小最大的范围。
  //  If the two parameters x_nMin and x_nMax are equal there are no limits.
  //  如果这两个参数x_nMin和x_nMax是相等的，那儿就不存在限制。
  //  After called this program, you will regenerate your interface.
  // 在call这个程序后，你会再生你的界面。
  //Input parameters  输入参数
  //  string x_sMsg : 字符串x_sMsg
  //    role : Message that you want to display 作用：你想去显示的消息
  //  num x_nItem : 数值量x_nItem
  //    role : Contains the value that you have enter 作用：包含你要去输入的值
  //  num x_nMin : 数值量x_nMin
  //    role : Limit minimum value 作用：最小值的限制
  //  num x_nMax : 数值量x_nMax
  //    role : Limit maximum value 作用：最大值的限制
  //
  //Example
  //  call insertDialog(scrMy,"Seconds :",l_nValue,0,10000)
  //
  //History
  //  Creation : 28-04-08 - f.Rob
  //  Modified : 08-08-11 - J.Cook     Changed $setTextMode to setTextMode
  //                                   And replaced literals ("", 0) with local variables
  //                                   when passing parameters by reference
  //
  //  Modified : 08-08-22 - J.Cook     Add screen parameter
  //Header end
  //-----------------------------------------------------------------------
  //Use for other task
  //If "insertDialog" is already used, put a message error and return in
  //如果"insertDialog"已经被使用，显示一个错误消息，在call程序的时候会返回
  //the calling program
  l_sEmpty = ""
  if watch(bShowDialog==false,2)==false
    bShowDialog=false
    logMsg("error dialog resoursing")
    return
  else
    setMutex(bShowDialog)
    call clear(x_scr, 0,13)
    l_sItem=toString("",x_nItem)
    call stringCopy(x_sMsg+">"+l_sItem,sMessage)
    //Divide the message if it is too long (Search a space for cut the message)
    //如果消息足够长，可以分割消息
    //Return the numbers of lines used for writing the message.
    //返回写入消息的行数
    call divideString(sMessage,l_nLine)
    l_nStartLine=round(5-l_nLine/2)
    //Start LINE
    call type(x_scr, 0,l_nStartLine-2,"┌──────────────────────────────────────┐")
    call type(x_scr, 0,l_nStartLine-1,"│                                      │")
    //Write the message
    for i=0 to l_nLine
      //Call type(,"                                      ")
      l_sMessage=sMessage[i]
      call typeCenter(x_scr, i+l_nStartLine,l_sMessage,38,false)
      call type(x_scr, 0,l_nStartLine+i,"│"+l_sMessage+"│")
    endFor
    //End LINE
    call type(x_scr, 0,l_nStartLine+l_nLine+1,"│                                      │")
    call type(x_scr, 0,l_nStartLine+l_nLine+2,"└──────────────────────────────────────┘")
    l_nPX=find(l_sMessage,">")+2
    l_nPY=l_nStartLine+l_nLine
    //Change the value
    call changeValue(x_scr, x_nItem,x_nMin,x_nMax,l_nPX,l_nPY,l_sEmpty)
    bShowDialog=false
    bUseRefresh=true
    delay(0)
  endIf
end

--- isListEmpty.pgx ---
public program isListEmpty(bool& x_bEmpty[])
begin
  //-----------------------------------------------------------------------
  //Header begin
  //Description of program
  //  Test if the list of Items is empty. 测试是否菜单列表为空
  //
  //Input parameters 输入参数
  //  bool x_bEmpty : 布尔量x_bEmpty
  //    role : Set to true if the list is empty and false otherwise
  //   作用：如果列表是空的，设为真值，否则返回假值。
  //Example
  //  call isListEmpty(l_bEmpty)
  //
  //History
  //  Creation : 28-04-08 - f.Rob
  //Header end
  //-----------------------------------------------------------------------
  if size(sItems)==1 and sItems[0]==""
    x_bEmpty=true
  else
    x_bEmpty=false
  endIf
end

--- leftPos.pgx ---
public program leftPos(string x_sItem, num x_nLength, string& x_sResult[])
  local num i
  local num l_nLength
  local string l_sItem
begin
  //-----------------------------------------------------------------------
  //Header begin
  //Description of program
  //  This program allows to keep x_nLength characters of a string from
  //  the left side.
  // 这个程序允许保留从左边开始计数的字符串中，x_nLength长度的字符。
  //  The characters after x_nLength on the right side will be truncated.
  // 在x_nLength长度右边的字符将会被截断。
  //Input parameters  输入参数
  //  string x_sItem : 字符串x_sItem
  //    role : string that you wan to cut 作用：你想去切割的字符串
  //  num x_nLength : 数值量x_nLength
  //    role : Length of the characters that you want to keep
  //    作用：你想去保留的字符
  //Output parameters 输出参数
  //  string x_sResult : 字符串x_sResult
  //    role : string truncated 作用：被截过后的字符串
  //
  //Example
  //  call leftPos("Staubli Robotics",7,sResult)
  //  put(sResult) //Displays "Staubli"
  //
  //History
  //  Creation : 28-04-08 - f.Rob
  //Header end
  //-----------------------------------------------------------------------
  l_sItem=x_sItem
  //Divide the string...
  if len(l_sItem)!=getDisplayLen(l_sItem) and x_nLength!=0
    for i=0 to len(x_sItem)-1
      l_nLength=l_nLength+getDisplayLen(left(l_sItem,1))
      l_sItem=right(l_sItem,len(l_sItem)-1)
      if l_nLength==x_nLength
        x_sResult=left(x_sItem,i+1)
        return
      else
        if l_nLength>x_nLength
          x_sResult=left(x_sItem,i)
          return
        endIf
      endIf
    endFor
  endIf
  x_sResult=left(x_sItem,x_nLength)
end

--- listAdd.pgx ---
public program listAdd(string& x_sItems[])
  local num i
  local num l_nSize
begin
  //Header begin
  //Description of program
  //  Insert x_sItems into the list.
  //  插入x_sItems进入到列表
  //Input parameters 输入参数
  //  string x_sItems : 字符串x_sItems
  //    role : Items to add  作用：要增加的条目
  //
  //Example
  //  call listAdd("Name: > ")
  //
  //History
  //  Creation : 28-04-08 - f.Rob
  //Header end
  for i=0 to (size(x_sItems)-1)
    if (size(sItems)!=1 or sItems!="") and x_sItems[i]!=""
      //Insert an Item in sItems[] after the last element.
      //在最后一个元素之后，在sItems[]插入一个条目。
      append(sItems)
      //Insert an Item in bReadWrite[] after the last element.
      //在最后一个元素之后，在bReadWrite[]插入一个条目
      append(bReadWrite)
    endIf
    if x_sItems[i]!=""
      sItems[size(sItems)-1]=x_sItems[i]
      //For default the RW is true
      bReadWrite[size(bReadWrite)-1]=true
    endIf
  endFor
end

--- listCreate.pgx ---
public program listCreate(screen& x_scr, string x_sTitle)
begin
  //-----------------------------------------------------------------------
  //Header begin
  //Description of program
  //  Create a list of data, displays the title x_sTitle,and draw
  //  the list from nTopX and nTopY position of the userPage (),
  //  of nBottomX length and height nBottomY.
  //  创建一个数据列表，显示x_sTitle的标题，然后画出列表的nTopX和nTopY位置在用户界面中，
  //  然后再画出长度nBottomX和高度nBottomY。
  //Input parameters  输入参数
  //  string x_Title : 字符串x_Title
  //    role : Title that you want for the list of data
  //   作用：你想要的数据列表的标题
  //Example
  //  Before using listCreate you can use setSizeList for defines all the
  //  parameters of position and size of the menu.
  // 在使用listCreate函数时，你能够先使用setSizeList来定义惨淡的位置和大小。
  //  call setSizeList(20,0,18,11)
  //  call listCreate(scrMy,"UserPage")
  //
  //History
  //  Creation : 28-04-08 - f.Rob
  //
  //  Modified : 08-08-22 - J.Cook     Add screen parameter
  //Header end
  //-----------------------------------------------------------------------
  sTitle=x_sTitle
  //Creation list of data
  call listFrame(x_scr,sTitle,nTopX,nTopY,nBottomX,nBottomY)
  call listEmpty()
end

--- listCursor.pgx ---
public program listCursor(screen& x_scr, num x_nView, bool x_bShow)
  local num l_nX
  local num l_nY
  local string l_sMessage
  local bool l_bEmpty
begin
  //-----------------------------------------------------------------------
  //Header begin
  //Description of program
  //  Place the cursor on the Item selected by x_nView and allows
  //  to inverse the video.
  //  将光变放在条目上选择x_nView，允许就是反相显示。
  //Input parameters  输入参数
  //  num x_nView : 数值量x_nView
  //    role : contains the Item selected  作用：包含已选的条目
  //  num x_bShow : 数值量x_bShow
  //    role : Allows to inverse video  作用：允许反相显示
  //    possible values : - true for inverse video  有可能的值：真值，当反相显示
  //                      - false font normal                   假值，当字体正常
  //
  //Example
  //  call listCursor(scrMy,2,l_bShow)
  //
  //History
  //  Creation : 28-04-08 - f.Rob
  //  Modified : 08-08-11 - J.Cook     Changed $setTextMode to setTextMode
  //                                   And replaced literals ("", 0) with local variables
  //                                   when passing parameters by reference
  //
  //  Modified : 08-08-22 - J.Cook     Add screen parameter
  //Header end
  //-----------------------------------------------------------------------
  call isListEmpty(l_bEmpty)
  if !l_bEmpty
    //The list is no empty
    nView=x_nView
    l_nX=nTopX+1
    l_nY=nTopY+1+x_nView
    if (nView+nFirst)>(size(sItems)-1)
      //Formatting the item depending on the width of the list (nBottomX)
      call strFill(sItems[size(sItems)-1],nBottomX,l_sMessage)
    else
      call strFill(sItems[nView+nFirst],nBottomX,l_sMessage)
    endIf
    gotoxy(x_scr, l_nX,l_nY)
    //Displays the Item
    if (x_bShow==true)
      //Inverse video
      setTextMode(x_scr, 1)
      put(x_scr, l_sMessage)
      setTextMode(x_scr, 0)
    else
      setTextMode(x_scr, 0)
      put(x_scr, l_sMessage)
    endIf
  endIf
end

--- listDel.pgx ---
public program listDel(num x_nIndex)
  local num l_nSize
begin
  //-----------------------------------------------------------------------
  //Header begin
  //Description of program
  //  Delete the element number x_nIndex of the list (sItems).
  //  删除列表（sItems）中的x_nIndex的元素数目
  //Example
  //  call listDel(3)
  //
  //History
  //  Creation : 28-04-08 - f.Rob
  //Header end
  //-----------------------------------------------------------------------
  l_nSize=size(sItems)-1
  //Test if the element number x_nIndex exist 测试x_nIndex元素数目是否存在
  if ((x_nIndex>=0) and (x_nIndex<=l_nSize))
    if l_nSize>0
      //Delete the element 删除元素
      delete(sItems[x_nIndex])
      delete(bReadWrite[x_nIndex])
    else
      sItems=""
      bReadWrite=true
    endIf
  endIf
end

--- listEmpty.pgx ---
public program listEmpty()
  local num i
  local num l_nSize
begin
  //-----------------------------------------------------------------------
  //Header begin
  //Description of program
  //  Delete all the elements of the list (sItems).
  //  删除列表（sItems）中的所有元素
  //Example
  //  call listEmpty()
  //
  //History
  //  Creation : 28-04-08 - f.Rob
  //Header end
  //-----------------------------------------------------------------------
  l_nSize=size(sItems)-1
  for i=0 to l_nSize
    if i>0
      //Destroy all elements of sItems 删除sItems中的所有元素
      delete(sItems[0])
      //Destroy all elements of bReadWrite  删除bReadWrite中的所有元素
      delete(bReadWrite[0])
    endIf
  endFor
  sItems=""
end

--- listEvent.pgx ---
public program listEvent(screen& x_scr, num x_nKey, num& x_nIndex[], string& x_sItem[])
  local num l_nSize
  local bool l_bEmpty
begin
  //-----------------------------------------------------------------------
  //Header begin
  //Description of program
  //  Read events from the keyboard and update the menu:  selected Items,
  //  cursor position.
  //  Return the selected Items and this name.
  //从键盘读取事件和更新菜单:选定的项目,光标位置。
  //返回选定的项目和名字。
  //Input parameters  输入参数
  //  num x_nKey : 数值量x_nKey
  //    role : Key pressed  作用：按键
  //Output parameters 输出参数
  //  num x_nIndex : 数值量x_nIndex
  //    role : Contains the number of the selected Item
  //    作用：包含已选条目的数目
  //  string x_sItem : 字符串x_sItem
  //    role : Contains the name of the selected Item
  //    作用：包含了已选条目的名字
  //Example
  //  call listEvent(scrMy,l_nKey,nIndex,sItem)
  //
  //History
  //  Creation : 28-04-08 - f.Rob
  //Header end
  //-----------------------------------------------------------------------
  call isListEmpty(l_bEmpty)
  if !l_bEmpty
    //The list is no empty  列表非空
    l_nSize=size(sItems)-1
    //Check the overFlow   检查溢出情况
    l_nSize=size(sItems)-1
    //Test if the selected element is in the list  测试是否已选元素在列表中
    if (nFirst+nView>l_nSize)
      //Reset the value 重设值
      nFirst=nView=0
    endIf
    //Security...
    switch (x_nKey)
      //Up
      case 261
        //Test if the cursor is not on the top of the menu  测试光标是否在菜单的顶部
        if ((nView-1)>=0)
          call listCursor(x_scr, nView,false)
          //Update the cursor of menu  更新菜单的光标
          nView=nView-1
          call listCursor(x_scr,nView,true)
          //Print the scroll  显示滚动条
        else
          if nView==0
            //Scrool up  滚动条置顶
            if ((nFirst-1)>=0)
              nFirst=nFirst-1
              //Move the Menu for obtain the Item number nFirst 移动菜单为的是获得在顶部的条目数
              //on the top
              call listUpdate(x_scr, nFirst)
            else
              //Go to the end of the menu  去菜单底部
              if nView+nFirst!=l_nSize
                call listCursor(x_scr, nView,false)
                call selectNewField(x_scr, l_nSize,nFirst+nView,nView)
              endIf
            endIf
          endIf
        endIf
      break
      //Down
      case 266
        //Test if the cursor is not on the bottom of the menu  测试光标是否在菜单的底部
        if ((nView+nFirst+1)<size(sItems))
          //No need to scrool only change cursor position  没有必要去滚动仅仅改变光标的位置
          if ((nView+1)<nBottomY)
            call listCursor(x_scr,nView,false)
            nView=nView+1
            call listCursor(x_scr,nView,true)
            //Print the scroll    显示滚动条
          else
            //Move UP
            nFirst=nFirst+1
            //Move the Menu for obtain the Item number nFirst  移动菜单为的是获得在顶部的条目数
            //on the top
            call listUpdate(x_scr,nFirst)
          endIf
        else
          //Go to the top of the menu 去到菜单的顶部
          if !(nView==0 and nFirst==0)
            call listCursor(x_scr,nView,false)
            nView=0
            call listUpdate(x_scr,0)
          endIf
        endIf
      break
      //Page Up  向上翻页
      case 262
        if !(nView==0 and nFirst==0)
          call listCursor(x_scr,nView,false)
          if ((nFirst+nView-nBottomY)>=0)
            //Move one page up 往上翻一页
            call selectNewField(x_scr,nFirst+nView-nBottomY,nFirst+nView,nView)
          else
            //Go to home  回到首页
            nView=0
            call listUpdate(x_scr,0)
          endIf
        endIf
      break
      //Page Down 向下翻页
      case 267
        if nView+nFirst!=l_nSize
          call listCursor(x_scr,nView,false)
          if ((nView+nFirst+nBottomY)<size(sItems)-1)
            //Move one page down   向下翻一页
            call selectNewField(x_scr,nFirst+nView+nBottomY,nFirst+nView,nView)
          else
            //Go to the end  到尾页
            call selectNewField(x_scr,l_nSize,nFirst+nView,nView)
          endIf
        endIf
      break
      //End
      case 269
        if nView+nFirst!=l_nSize
          //Move to end  移动到末尾
          call listCursor(x_scr,nView,false)
          call selectNewField(x_scr,l_nSize,nFirst+nView,nView)
        endIf
      break
      //Home
      case 265
        if !(nView==0 and nFirst==0)
          //Move to home  回首页
          call listCursor(x_scr,nView,false)
          nView=0
          call listUpdate(x_scr,0)
        endIf
      break
      default
      break
    endSwitch
    x_nIndex=nFirst+nView
    x_sItem=sItems[x_nIndex]
  endIf
end

--- listFrame.pgx ---
program listFrame(screen& x_scr, string x_sTitle, num x_nX, num x_nY, num x_nDx, num x_nDy)
  local num l_nDx
  local num l_nDy
  local num i
  local string l_sStr
  local string l_sStrLine
  local num l_nValue
begin
  //-----------------------------------------------------------------------
  //Header begin
  //Description of program
  //  Create a list of data, displays the title sTitle, and draw the list
  //  to the position pX and pY of the userPage (), of pDX length and height
  //  pDY.
  // 创建数据的列表，显示标题sTitle，画出用户界面的原点位置pX和pY上，长度和高度为pDX和pDY
  //Input parameters  输入参数
  //  num x_nX : 数值量x_nX
  //    role : cursor column position : top left corner for the beginning of the list menu
  //    作用：光标列的位置：左上角开始菜单列表
  //  num x_nY : 数值量x_nY
  //    role : cursor row position : top left corner for the beginning of the list menu
  //    作用：光标行的位置：左上角开始菜单列表
  //  num x_nDx : 数值量x_nDx
  //    role : width of the box  作用：用户界面的宽度
  //  num x_nDY : 数值量x_nDY
  //    role : height of the box  作用：用户界面的高度
  //
  //Example
  //  call listFrame(scrMy,"UserPage",20,0,18,11)
  //
  //History
  //  Creation : 28-04-08 - f.Rob
  //
  //  Modified : 08-08-22 - J.Cook     Add screen parameter
  //Header end
  //-----------------------------------------------------------------------
  l_sStrLine="─────────────────────────────────────────"
  l_nDx=x_nDx
  l_nDy=x_nDy
  //Top
  //Cut the l_sStrLine at the width l_nDx
  l_sStr="┌"+mid(l_sStrLine,l_nDx,0)+"┐"
  //Displays the top line
  gotoxy(x_scr, x_nX,x_nY)
  put(x_scr, l_sStr)
  l_nValue=x_nX+2
  //Title
  if x_sTitle!=""
    call leftPos("┤"+x_sTitle+"├",l_nDx,x_sTitle)
    gotoxy(x_scr, x_nX+l_nDx-getDisplayLen(x_sTitle)+1,x_nY)
    put(x_scr, x_sTitle)
  endIf
  //Containt
  for i=1 to l_nDy
    l_nValue=x_nY+i
    l_sStr="│"
    gotoxy(x_scr, x_nX,l_nValue)
    put(x_scr, l_sStr)
    gotoxy(x_scr, x_nX+l_nDx+1,l_nValue)
    put(x_scr, l_sStr)
  endFor
  //Bottom
  l_nValue=x_nY+i
  //Cut the l_sStrLine at the width l_nDx
  l_sStr="└"+mid(l_sStrLine,l_nDx,0)+"┘"
  //Displays the bottom line
  gotoxy(x_scr, x_nX,l_nValue)
  put(x_scr, l_sStr)
end

--- listins.pgx ---
public program listIns(string& x_sItems[], num x_nPos)
  local num i
  local num l_nSize
begin
  //-----------------------------------------------------------------------
  //Header begin
  //Description of program
  //  Insert an element x_sItem before the number x_nPos.
  //  插入一个元素x_sItem在x_nPos位置之前
  //Input parameters 输入参数
  //  num x_nPos :  数值量x_nPos
  //    role : Position in the array sItems where you want to insert an new Item
  //    作用：在数组sItems的某个位置，你想插入一个新条目
  //Output parameters  输出参数
  //  string x_sItem : 字符串x_sItem
  //    role : Item that you want to insert
  //   作用：你想去插入的条目
  //Example
  //  call listIns("Staubli",3)
  //
  //History
  //  Creation : 28-04-08 - f.Rob
  //Header end
  //-----------------------------------------------------------------------
  l_nSize=size(sItems)-1
  //Test if the position x_nPos is in the array 测试是否这个位置在数组中
  if ((x_nPos>=0) and (x_nPos<=l_nSize))
    for i=0 to (size(x_sItems)-1)
      if size(sItems)!=1 or sItems!=""
        //Insert an element in sItems[] 插入一个元素到sItems[]
        insert(sItems[x_nPos+i])
        insert(bReadWrite[x_nPos+i])
      endIf
      sItems[x_nPos+i]=x_sItems[i]
      //For default the RW is true 默认是RW为真
      bReadWrite[x_nPos+i]=true
    endFor
  else
    //Position not in the array 位置没有在数组中
    //Insert the element 插入元素
    call listAdd(x_sItems)
  endIf
end

--- listRedraw.pgx ---
public program listRedraw(screen& x_scr, num x_nFirst)
begin
  //-----------------------------------------------------------------------
  //Header begin
  //Description of program
  //  Redraw the list in the userPage from the element number.
  //  pFirst of the list.
  //  重画在用户界面的pFirst列表的元素数目
  //Input parameters  输入参数
  //  num x_nFirst :  数值量x_nFirst
  //    role : Defines the first element of the list
  //    作用：定义列表的第一个元素
  //Example
  //  call listRedraw(scrMy,1)
  //
  //History
  //  Creation : 28-04-08 - f.Rob
  //
  //  Modified : 08-08-22 - J.Cook     Add screen parameter
  //Header end
  //-----------------------------------------------------------------------
  call listFrame(x_scr, sTitle,nTopX,nTopY,nBottomX,nBottomY)
  call listUpdate(x_scr, x_nFirst)
end

--- listUpdate.pgx ---
public program listUpdate(screen& x_scr, num x_nFirst)
  local num i
  local num l_nLen
  local string l_sStr
  local string l_sStr2
  local num l_nValue
  local num l_nView
  local num l_nX
  local num l_nY
  local num l_nSize
  local bool l_bEmpty
begin
  //-----------------------------------------------------------------------
  //Header begin
  //Description of program
  //  Update the menu : moves the list to obtain the Item number x_nFirst
  //  on the top.
  // 更新菜单：移动到列表来获得x_nFirst的条目数。
  //Input parameters  输入参数
  //  num x_nFirst : 数值量x_nFirst
  //    role : Element on the top of the menu
  //   作用：菜单顶部的元素
  //Example
  //  call listUpdate(scrMy,0) //put the Item 0 on the top of the list
  //
  //History
  //  Creation : 28-04-08 - f.Rob
  //
  //  Modified : 08-08-22 - J.Cook     Add screen parameter
  //Header end
  //-----------------------------------------------------------------------
  if x_nFirst>=0
    nFirst=x_nFirst
  else
    nFirst=0
  endIf
  //Save the coordinate
  l_nValue=nBottomY-1
  //Check the overFlow
  l_nSize=size(sItems)-1
  if (nFirst+nView>l_nSize)
    //Reset the value
    nFirst=nView=0
  endIf
  i=0
  //Check the unKnow problem
  if l_nSize<l_nValue
    if nFirst!=0
      nView=nView+nFirst
      nFirst=0
    endIf
  endIf
  do
    l_nX=nTopX+1
    l_nY=nBottomY+i-1
    l_nY=nTopY+i+1
    l_nLen=nBottomX
    if ((i+nFirst)<size(sItems))
      //Print the item
      if (l_nSize>=0)
        l_sStr=mid(sItems[(i+nFirst)],l_nLen,0)
      endIf
    else
      //Print the blank line
      l_sStr="                                        "
    endIf
    //Fill the line
    call strFill(l_sStr,l_nLen,l_sStr2)
    gotoxy(x_scr, l_nX,l_nY)
    put(x_scr, l_sStr2)
    i=i+1
  until (i>l_nValue)
  //Underline the actual line
  call isListEmpty(l_bEmpty)
  if !l_bEmpty
    call listCursor(x_scr, nView,true)
  else
    call listCursor(x_scr, nView,false)
    nView=0
    nFirst=0
  endIf
  //Print the scroll
  call printScroll(x_scr)
  //Leave the resourse
  delay(0)
end

--- midPos.pgx ---
public program midPos(string x_sItem, num x_nLength, num x_nPos, string& x_sResult[])
  local string l_sLeft
begin
  //-----------------------------------------------------------------------
  //Header begin
  //Description of program
  //  This program allows to keep x_nLength characters of a string from
  //  a position x_nPos.
  // 该程序允许保留一个字符串中x_nPos位置开始的 x_nLength长度的字符。
  //  The characters before and after x_nPos and x_nPos+x_nLength will be
  //  truncated.
  //  字符在x_nPos之前和x_nPos+x_之后的字符都会被截断。
  //Input parameters  输入参数
  //  string x_sItem :  字符串x_sItem
  //    role : string that you wan to cut 作用：你想去切分的字符串
  //  num x_nLength : 数值量x_nLength
  //    role : Length of the characters that you want to keep  作用：你想要去保留的字符长度
  //  num x_nPos :  数值量x_nPos
  //    role : Position to start keeping characters
  //  作用：开始保留字符的位置
  //Output parameters 输出参数
  //  string x_sResult : 字符串x_sResult
  //    role : string truncated
  //   作用：截断后的字符串
  //Example
  //  call midPos("Staubli Robotics",4,2,sResult)
  //  put(sResult) //Displays "aubl"
  //
  //History
  //  Creation : 28-04-08 - f.Rob
  //Header end
  //-----------------------------------------------------------------------
  // LEFT SIDE
  call leftPos(x_sItem,x_nLength+x_nPos,l_sLeft)
  // update
  x_sResult=l_sLeft
  // RIGHT SIDE
  call rightPos(l_sLeft,x_nLength,x_sResult)
  // OK ....
end

--- nullKey.pgx ---
public program nullKey(screen& x_scr, num& x_nKey[])
begin
  //-----------------------------------------------------------------------
  //Header begin
  //  Wait a new key was pressed, and put x_nKey to 0.
  //  等待一些按键后，放x_nKey到0
  //  This program was used for waiting the release of a button.
  // 这个程序被用来去等待按键的释放
  //Input parameter  输入参数
  //  num x_nKey :  数值量x_nKey
  //    role : this variable is put to 0 when a new key was pressed.
  //    作用：当一个新按键被按后，这个变量回到0
  //Example
  //  call nullKey(scrMy,l_nKey)
  //
  //History
  //  Creation : 28-04-08 - f.Rob
  //
  //  Modified : 22 Aug 2011 - J. Cook  Added user screens
  //Header end
  //-----------------------------------------------------------------------
  //Wait a new key stroke
  wait(getKey(x_scr)==-1)
  x_nKey=0
end

--- numCopy.pgx ---
public program numCopy(num& x_nCopy[], num& x_nPaste[])
// Copy all the value from the x_nCopy to x_nPaste
  local num i
  local num l_nSize
begin
  //-----------------------------------------------------------------------
  //Header begin
  //Description of program
  //  Copy all the values from x_nCopy to x_nPaste.
  //  You can copy an array of numerical values.
  //  复制所有的变量重x_nCopy到x_nPaste
  //  你能够复制一个数值量的数组
  //Input parameters  输入参数
  //  num x_nCopy :数值量 x_nCopy
  //    role : Value(s) that you want to copy
  //    作用：你想要去复制的值
  //  num x_nPaste :数值量x_nPaste
  //    role : Value(s) paste
  //    作用：要去粘贴的值
  //Example
  //  call numCopy("641",nPaste) //nPaste=641 at the end of the program
  //
  //History
  //  Creation : 28-04-08 - f.Rob
  //
  //  Modified : 08-08-22 - J.Cook     Add screen parameter
  //Header end
  //-----------------------------------------------------------------------
  //Copy all the value from the first element to the second one
  l_nSize=size(x_nPaste)
  if size(x_nCopy)>size(x_nPaste)
    //Redim the Paste String ARRAY
    for i=l_nSize to (size(x_nCopy)-1)
      insert(x_nPaste[i])
    endFor
  else
    if size(x_nCopy)<size(x_nPaste)
      for i=size(x_nCopy) to l_nSize-1
        delete(x_nPaste[size(x_nCopy)])
      endFor
    endIf
  endIf
  //Copy all the field
  for i=0 to (size(x_nCopy)-1)
    x_nPaste[i]=x_nCopy[i]
  endFor
end

--- printScroll.pgx ---
program printScroll(screen& x_scr)
  local num i
  local num lX
  local num lY
begin
  //-----------------------------------------------------------------------
  //Header begin
  //Description of program
  //  Put the scrool on the right of the list menu.
  // 在列表菜单右边放滚动条
  //History
  //  Creation : 28-04-08 - f.Rob
  //
  //Example
  //  call printScroll(scrMy)
  //
  //  Modified : 08-08-22 - J.Cook     Add screen parameter
  //Header end
  //-----------------------------------------------------------------------
  if size(sItems)>nBottomY
    //Find the percentage
    //Windows style
    //i=(size(sItems)-nBottomY+1)/(nFirst+1)
    // nokia style
    i=(size(sItems))/(nFirst+nView+1)
    lX=nTopX+nBottomX+1
    lY=roundUp((nBottomY)/i+nTopY)
    for i=nTopY+1 to nBottomY
      gotoxy(x_scr, lX,i)
      if i==lY
        //
        put(x_scr, "■")
        //
      else
        put(x_scr, "│")
      endIf
    endFor
  endIf
end

--- questionDialog.pgx ---
public program questionDialog(screen& x_scr, string x_sMsg, string& x_sButton[], num& x_nResult[])
  local bool lExit
  local num nLine
  local num i
  local num nStartLine
  local string l_sMessage
begin
  //-----------------------------------------------------------------------
  //Header begin
  //Description of program
  //  Displays a dialog box with a confirm question.
  //  Possibility to add buttons on the menu.
  //  After called this program, you will regenerate your interface.
  //  显示一个是否确认的对话框，有可能在菜单上增加按键，在call这个程序后，你可以再生界面。
  //Input parameters  输入参数
  //  string x_sMsg :  字符串x_sMsg
  //    role : Message that you want to displays in the dialog box
  //    作用：你想要去显示在对话框里的消息
  //Output parameter  输出参数
  //  string x_sButton  字符串x_sButton
  //    role : Button(s) that you want to display. Possibility to displays up to
  //    作用：你想要去显示的按键，有可能用到八个键（F1 到 F8）
  //    8 buttons (F1 to F8).
  //  num x_nResult : 数值量x_nResult
  //    role : Contains the number of the key pressed
  //    作用：包含按键的数值
  //    posssible values : 0  => ENTER
  //                       -1 => ESC
  //                       1  => F8
  //                       2  => F7
  //                        ...
  //                       8  => F1
  //
  //Example
  //  l_sButton="Yes"
  //  l_sButton[1]="No"
  //  call questionDialog(scrMy,"Do you want to quit a program ?",l_sButton,l_nKey)
  //
  //History
  //  Creation : 28-04-08 - f.Rob
  //
  //  Modified : 08-08-22 - J.Cook     Add screen parameter
  //Header end
  //-----------------------------------------------------------------------
  //Use for other task
  //If questionDialog is already used, put a message error and return in
  //the calling program
  if watch(bShowDialog==false,2)==false
    bShowDialog=false
    logMsg("error dialog resoursing")
    return
  else
    setMutex(bShowDialog)
    if x_sMsg!=""
      call stringCopy(x_sMsg,sMessage)
      //Divide the message if it is too long (Search a space for cut the message)
      //Return the numbers of lines used for writing the message.
      call divideString(sMessage,nLine)
      nStartLine=round(5-nLine/2)
      //Start LINE
      call type(x_scr, 0,nStartLine-2,"┌──────────────────────────────────────┐")
      call type(x_scr, 0,nStartLine-1,"│                                      │")
      //Write the message
      for i=0 to nLine
        l_sMessage=sMessage[i]
        call typeCenter(x_scr, i+nStartLine,l_sMessage,38,false)
        call type(x_scr, 0,nStartLine+i,"│"+l_sMessage+"│")
      endFor
      //End LINE
      call type(x_scr, 0,nStartLine+nLine+1,"│                                      │")
      call type(x_scr, 0,nStartLine+nLine+2,"└──────────────────────────────────────┘")
    endIf
    //Write the button message
    call clear(x_scr, 0,13)
    for i=0 to size(x_sButton)-1
      call typeMenu(x_scr, 8-i,x_sButton[i])
    endFor
    lExit=false
    x_nResult=-100
    do
      nKey=get(x_scr)
      switch (nKey)
        //Enter
        case 270
          x_nResult=0
        break
        //ESC
        case 255
          x_nResult=-1
          bUseEscape=true
        break
        default
          //Look if the button press is defined
          if (nKey>=271 and nKey<=278) and ((279-nKey)<=size(x_sButton))
            if x_sButton[278-nKey]!=""
              x_nResult=279-nKey
            endIf
          endIf
        break
      endSwitch
      delay(0)
    until (x_nResult!=-100)
    call nullKey(x_scr,nKey)
    //Release
    bShowDialog=false
    bUseRefresh=true
  endIf
end

--- read.pgx ---
public program read(screen& x_scr, num x_nX, num x_nY, string& x_sMsg[], num x_nLength, bool x_bCrypt)
// Read one string from the pX column and pY line
  local num l_nLength
  local bool l_bExit
  local bool l_bBlk
  local num i
  local num p
  local num l_nTps
  local string l_sMsg
  local string l_sView
  local string l_sStr
begin
  //-----------------------------------------------------------------------
  //Header begin
  //Description of program
  //  Get a message limited to x_nLength and write it on the pX column
  //  and pY line.
  //  得到一条消息长度限制在 x_nLength内，把它写到pX列pY行。
  //  If x_bCrypt is true all the characters displayed will be replaced by "*",
  //  otherwise by the corresponding characters.
  // 如果x_bCrypt是真的，显示的所有字符将会被"*"替代，否则就用相应的字符替代。
  //  The message is validate by "ENTER" key. "ESC" or "F1 to F8"
  //  消息是由回车键确认，ESC键火车F1到F8键取消输入，消息将会恢复到初始状态。
  //  keys cancel value, the message will resume this initial value.
  //
  //Input parameters
  //  num x_nX : 数值量x_nX
  //    role : Cursor column
  //    作用：光标列
  //    possible values : 0 to 39
  //    可能的值：0到39
  //  num x_nY : 数值量x_nY
  //    role : Cursor row
  //    作用:光标行
  //    possible values : 0 to 13  可能的值：0到13
  //  num x_nLength : 数值量x_nLength
  //    role : limit the lenght of the message
  //    作用：限制消息的长度
  //  bool x_bCrypt :  布尔量x_bCrypt
  //    role : crypt the message that you are seized
  //    作用：你要抓住的消息
  //    possibles values : true => crypt the message
  //                       false => writing normal
  //
  //Output parameters 输出参数
  //  string x_sMsg :  字符串x_sMs
  //    role : Message reading  作用：读取的消息
  //
  //Example
  //  call read(scrMy,15,7,l_sItem,10,false)
  //
  //History
  //  Creation : 28-04-08 - f.Rob
  //  Modified : 08-08-11 - J.Cook     Changed $setTextMode to setTextMode
  //                                   And replaced literals ("", 0) with local variables
  //                                   when passing parameters by reference
  //
  //  Modified : 08-08-22 - J.Cook     Add screen parameter
  //Header end
  //-----------------------------------------------------------------------
  l_nTps=clock()
  l_sMsg=x_sMsg
  p=len(l_sMsg)
  //Cryptage
  if x_bCrypt
    do
      i=len(l_sMsg)
      nKey=getKey(x_scr)
      if ((clock()-l_nTps)>=0.5)
        if l_bBlk==true
          l_bBlk=false
        else
          l_bBlk=true
        endIf
        l_nTps=clock()
      endIf
      if (nKey>=32) and (nKey<=126)
        if ((len(l_sMsg)+1)<=x_nLength)
          l_sMsg=l_sMsg+chr(nKey)
        endIf
      else
        //Backspace
        if (nKey==263) and (len(l_sMsg)>0)
          l_sMsg=mid(l_sMsg,len(l_sMsg)-1,0)
        endIf
      endIf
      if (l_sStr!=l_sMsg)
        call strFillChr(l_sMsg,l_sView,"*")
        l_sStr=l_sMsg
      endIf
      if l_bBlk==true
        call typeLen(x_scr, x_nX,x_nY,l_sView+"|",x_nLength+1)
      else
        call typeLen(x_scr, x_nX,x_nY,l_sView+" ",x_nLength+1)
      endIf
      //Release the resource
      delay(0)
    until (nKey==270) or (nKey==255)
  else
    //Normal read
    //Delete the old value
    setTextMode(x_scr, 0)
    call strFillChr(l_sMsg,l_sView," ")
    call typeLen(x_scr, x_nX,x_nY,l_sView,40-x_nX-1)
    //Read the new one
    gotoxy(x_scr, x_nX,x_nY)
    get(x_scr, l_sMsg)
  endIf
  //Save the escape key pressure
  if isKeyPressed(x_scr, 255)
    bUseEscape=true
  else
    bUseEscape=false
  endIf
  //Result
  if (isKeyPressed(x_scr, 270) or nKey==270 or l_sMsg!=x_sMsg) and !bUseEscape
    x_sMsg=l_sMsg
  endIf
end

--- readme.pgx ---
program readme()
begin
  //Title : Teach pendant based user interface tools
  //
  //General description :
  //  This library provides tools to assist in the implementation of a
  //  teach pendant based semi-graphical user interface in VAL3.
  //  This manager provides programs allowing to display, enter data or manage a list
  //  of data in the userPage () of the CS8.
  // 这个库提供工具来协助实现示教器上的基于VAL3语言的半图形化用户界面。
  //  管理人员可以提供程序使显示,输入数据或管理一个数据列表在CS8的用户界面上。
  //
  //Hardware required :  硬件需要
  //  - Robot system    : any Staubli robot  机器人系统：任何Staubli机器人
  //  - Peripherals     : no peripherals required  外设：不需要外设
  //
  //VAL3 options :  VAL3选项
  //  - VAL3 version    : 7.1.3   VAL3版本：7.1.3
  //  - VAL3 licenses   : PaintiXen or VALPlast in demo mode   VAL3 许可证：演示模式的PaintiXen或者VALPlast
  //  - VAL3 add-ons    : none    VAL3 add-ons：没有
  //
  //Library version     : 7.1.2.0   库版本：7.1.2.0
  //
  //Public variables    :  公共变量
  //  - bool bShowDialog : Set to true during every displaying of a dialog window :
  //    insertDialog(), questionDialog(), timerDialog(). You can't run two dialogs
  //    window at the same time.
  //    布尔量bShowDialog：在每次显示一个对话框窗口：insertDialog(), questionDialog(), timerDialog()
  //    设置为真值。你不能同时运行两个窗口。
  //  - bool bUseEscape : set to true when you press ESC and false otherwise.
  //    This value is updating in several programs which use a user dialog.
  //    布尔量bUseEscape：当你按ESC键的时候，设置为真，否则为假。
  //    这个值会在几个程序使用同一个用户窗口的时候更新。
  //  - bool bUseRefresh : Set to true after every displaying of a dialog window :
  //    insertDialog(), questionDialog(), setView(), timerDialog().
  //    布尔量bUseRefresh：在每次显示一个对话框窗口时，设为真值：insertDialog(), questionDialog(), setView(), timerDialog()
  //    When you use several tasks you must do a refresh.
  //    当你在使用许多任务时，你必须做一个刷新。
  //  - num nBottomX, nBottomY, nTopX, nTopY : position of the list menu. (See setSizeList())
  //    数值量nBottomX, nBottomY, nTopX, nTopY：列表菜单的位置（看setSizeList()）
  //  - num nPage : Utilisation to know the current page which is open.
  //    You could use it when you have several pages.
  //    数值量nPage：可以知道当前哪个页面是打开的。当你有许多页面时，你可以使用它。
  //  - num nView : Give the current position of the list cursor : if you use a list with a size
  //    of 10 elements the current position is between 0 to 10
  //    数值量nView：给予目前列表光标的位置：如果你使用的列表大小为10个元素，那么目前的位置在0到10之间。
  //    (different that the position of the selected Items)
  //  - string sItems : This array of string, contains the list of the current data.
  //    字符串sItems：字符串的数组，包含了当前数据的列表。
  //Included libraries  : none  包含的库：没有
  //
  //Miscellaneous       : ---   杂项;---
  //
  //Keywords            : GUI, manager, interface, gestionnaire, user interface,
  //                    interface utilisateur, list, liste, human-machine, homme-machine
  //                    semi-graphical, semi-graphique
  //关键词：用户图形界面、管理员、使用界面的用户,列表,人机交互,半图形化
  //
end

--- rightPos.pgx ---
public program rightPos(string x_sItem, num x_nLength, string& x_sResult[])
  local num i
  local num l_nLength
  local string l_sItem
begin
  //-----------------------------------------------------------------------
  //Header begin
  //Description of program
  //  This program allows keeping x_nLength characters of a string from
  //  the right side.
  //  The characters after x_nLength on the left side will be truncated.
  //  这个程序允许从右边数起保留x_nLength长度的字符。在x_nLength长度左边的字符会被截断。
  //Input parameters  输入参数
  //  string x_sItem : 字符串x_sItem：
  //    role : string that you wan to cut  作用：你想去分割的字符串
  //  num x_nLength : 数值量x_nLength：
  //    role : Length of the characters that you want to keep
  //   作用：你想去保留的字符长度
  //Output parameters  输出参数
  //  string x_sResult :  字符串x_sResult
  //    role : string truncated  作用：被截断的字符串
  //
  //Example
  //  call leftPos("Staubli Robotics",8,sResult)
  //  put(sResult) //Displays "Robotics"
  //
  //History
  //  Creation : 28-04-08 - f.Rob
  //Header end
  //-----------------------------------------------------------------------
  l_sItem=x_sItem
  //Divide the string...
  if len(l_sItem)!=getDisplayLen(l_sItem) and x_nLength<=getDisplayLen(l_sItem)
    for i=len(x_sItem)-1 to 0 step -1
      l_nLength=l_nLength+getDisplayLen(right(l_sItem,1))
      l_sItem=left(l_sItem,len(l_sItem)-1)
      if l_nLength==x_nLength
        x_sResult=right(x_sItem,len(x_sItem)-i)
        return
      else
        if l_nLength>x_nLength
          x_sResult=right(x_sItem,len(x_sItem)-i-1)
          return
        endIf
      endIf
    endFor
  endIf
  x_sResult=right(x_sItem,x_nLength)
end

--- selectNewField.pgx ---
public program selectNewField(screen& x_scr, num x_nSelected, num x_nIndex, num x_nView)
  local num l_nFirst
begin
  //-----------------------------------------------------------------------
  //Header begin
  //Description of program
  //  Select a new item with a user friendly system.
  //  Usually use when you create a new Item and you want to select it.
  //  This program update the list with the the element x_nSelected
  //  that you want to selected.
  //  选择与用户交互性友好系统的一个新条目
  //  当你去创建一个新条目，你想去选择它时，常常会使用
  //  该程序更新了你想去选择的元素x_nSelected列表。
  //Input parameters  输入参数
  //  num x_nSelected : 数值量x_nSelected
  //    role : position that you want to go in the list
  //    作用：你想去到的列表的位置
  //    possible values : - "-1" : place current selected element in the
  //    middle of the list.
  //                      - other values : place the element in the middle of the list.
  //    有可能的值：- "-1" ：放置目前已选的元素在列表的中部。
  //  num x_nIndex :
  //    role : current position in the list
  //    作用：列表中目前位置
  //  num x_nView :
  //    role : current position of the list cursor
  //    作用：列表光标目前的位置
  //Examples
  //  call selectNewField(scrMy,7,4,3)  //Displays the Item number 7 in the
  //                              middle of the list
  //  call selectNewField(scrMy,-1,7,4) //Place the current selected Item
  //                              in the middle of the list
  //
  //History
  //  Creation : 28-04-08 - f.Rob
  //
  //  Modified : 08-08-22 - J.Cook     Add screen parameter
  //Header end
  //-----------------------------------------------------------------------
  // Update the first value from the parameter
  l_nFirst=max(x_nIndex-x_nView,0)
  // Do only an update of the first item
  if (x_nSelected==-1)
    nView=x_nView
    call listUpdate(x_scr, x_nIndex-x_nView)
  else
    //Select the new field using a scroll logic
    //The new value is not in the screen
    if x_nSelected<l_nFirst or abs(x_nSelected-l_nFirst)>=(nBottomY)
      //Start from the beginnnig
      if x_nSelected<l_nFirst and x_nSelected<nBottomY
        nView=x_nSelected
        call listUpdate(x_scr, 0)
      else
        if x_nSelected<size(sItems)-nBottomY
          //Move the list and select the field in the middle
          nView=roundUp(nBottomY/2)
        else
          nView=x_nSelected-(size(sItems)-nBottomY)
        endIf
        call listUpdate(x_scr, abs(x_nSelected-nView))
      endIf
    else
      //Move only the nView of the field
      nView=abs(x_nSelected-l_nFirst)
      call listUpdate(x_scr, abs(x_nIndex-x_nView))
    endIf
  endIf
end

--- setMenu.pgx ---
public program setMenu(screen& x_scr, string& x_sMenuName[], bool x_bShowName, num x_nY)
  local num i
begin
  //-----------------------------------------------------------------------
  //Header begin
  //Description of program
  //  Displays a menu from an array of string.
  //  Every elements of the array defines the name of one Item of the menu.
  //  The first element defines F1, the second F2...,
  //  You MUST pass an array with a size 8.
  //  从一个字符串数组中显示一个菜单。
  //  数组中的每个元素定义了菜单中每个条目的名字。
  //  第一个元素定义为F1，第二个为F2...,
  //  你必须通过一个大小为8的数组
  //Input parameters
  //  bool x_bShowName :
  //    role : For show the names of the functions key on the bottom side.
  //    作用：在底部展示函数的名字
  //    possible values : true  => displays the names of the functions
  //                      false => displays F1 to F8
  //    有可能的值：真值=>显示函数名
  //                假值=>显示F1 to F8
  //  num x_nY :
  //    role : Cursor row for start the menu
  //   作用：光标行去开始菜单
  //Outup parameters
  //  string x_sMenuName :
  //    role : It's an array of string, every elements represent an Item for the
  //    menu.
  //   作用：这是一个字符串数组，每一个元素代表菜单的一个条目
  //Example
  //  Before using setMenu you can use stringToArray for an easy utilisation :
  //  l_sMenu="Exit,Clear,,,,Del,Add,Ins"
  //  call stringToArray(l_sMenu,sMenu)
  //  call setMenu(scrMy,sMenu,true,3)
  //
  //History
  //  Creation : 28-04-08 - f.Rob
  //  A
  //  Modified : 08-08-22 - J.Cook   dd screen parameter
  //Header end
  //-----------------------------------------------------------------------
  if size(x_sMenuName)<9
    //Size x_sMenuName ok
    for i=0 to (size(x_sMenuName)-1)
      if x_sMenuName[i]!="" and x_sMenuName[i]!=" "
        if x_bShowName==false
          //Replace user text by F1, F2...
          call typeMenu(x_scr, i+1,"F"+toString("1",i+1))
        else
          //Displays menu
          call typeMenu(x_scr,i+1,x_sMenuName[i])
        endIf
        if x_nY!=-1
          //x_nY ok : menu start in the screen
          call type(x_scr,0,i+x_nY,("F"+(toString("1",i+1)+" "+x_sMenuName[i])))
        endIf
      endIf
    endFor
  endIf
end

--- setSizeList.pgx ---
public program setSizeList(num x_nPx, num x_nPy, num x_nPBottomX, num x_nPBottomY)
begin
  //-----------------------------------------------------------------------
  //Header begin
  //Description of program
  //  Defines all the parameters of positions and size of the list menu.
  // 定义列表菜单中所有参数的位置和大小
  //Input parameters
  //  num x_nPx:
  //    role : cursor column position : top left corner for the beginning of
  //    the list menu
  //    作用：光标列位置：在列表菜单开始的左上角
  //  num x_nPy :
  //    role : cursor column position : top left corner for the beginning of
  //    the list menu
  //    作用：光标行位置：在列表菜单的开始的左上角
  //  num x_nPBottomX
  //    role : width of the box
  //    作用：窗口的宽度
  //  num x_nPBottomY :
  //    role : height of the box
  //    作用：窗口的高度
  //Example
  //  call setSizeList(20,0,18,11)
  //
  //History
  //  Creation : 28-04-08 - f.Rob
  //Header end
  //-----------------------------------------------------------------------
  //Put all the parameters in globals variables
  nTopX=nTopX[1]=x_nPx
  nTopY=x_nPy
  nBottomX=nBottomX[1]=x_nPBottomX
  nBottomY=x_nPBottomY
end

--- setView.pgx ---
public program setView(bool x_bLarge)
begin
  //-----------------------------------------------------------------------
  //Header begin
  //Description of program
  //  Allows enlarging the width of the list menu. After called this
  //  program, you will regenerate your interface.
  //  允许扩大列表菜单的宽度。在call了这个程序后，你将会重生你的界面。
  //Input parameters
  //  bool x_bLarge :
  //    role : For enlarge the width of the list menu. 为了扩大列表才菜单的宽度。
  //    posssible value : true  => enlarge the width of the list menu
  //                      false => normal width (width defines with setSizeList)
  //
  //Example
  //  call x_bLarge(true)
  //
  //History
  //  Creation : 28-04-08 - f.Rob
  //Header end
  //-----------------------------------------------------------------------
  //Save the TopX position in an other element
  //Put TopX width on the maximum (38) for enlarge the list menu
  if x_bLarge
    nTopX[1]=nTopX
    nTopX=0
    nBottomX[1]=nBottomX
    nBottomX=38
  else
    //Restore the TopX position saved
    nTopX=nTopX[1]
    nBottomX=nBottomX[1]
  endIf
  bUseRefresh=true
end

--- showBoolStatus.pgx ---
public program showBoolStatus(bool x_bStatus, string& x_sEvent[])
begin
  //-----------------------------------------------------------------------
  //Header begin
  //Description of program
  // Add a character "x" in x_sEvent if a x_bStatus bool value is true.
  // 如果x_bStatus布尔值是真的，增加一个字符"x" 到x_sEvent中。
  //Input parameters
  //  bool x_bStatus :
  //    role : Add the character of status.
  //    作用：增加字符的状态
  //    possible values : true => add character x
  //    有可能的值：真 => 增加字符x
  //Output parameters
  //  string x_sEvent :
  //    role : string returned
  //    作用：返回的字符串
  //    possible values : When x_bStatus->true  => x_sEvent -> [x]
  //                      When x_bStatus->false => x_sEvent -> [ ]
  //    有可能的值：当x_bStatus->为真=>x_sEvent -> [x]
  //                当x_bStatus->为假=> x_sEvent -> [ ]
  //Example
  //  call showBoolStatus(bStatus,sEvent)
  //
  //History
  //  Creation : 28-04-08 - f.Rob
  //Header end
  //-----------------------------------------------------------------------
  if x_bStatus
    x_sEvent="[x]"
  else
    x_sEvent="[ ]"
  endIf
end

--- strFill.pgx ---
public program strFill(string x_sMessageIn, num x_nLenMessOut, string& x_sMessageOut[])
  local string l_sEmpty
  local num l_nLen
begin
  //-----------------------------------------------------------------------
  //Header begin
  //Description of program
  //  To add spaces if the length of x_sMessageIn is less than the
  //  x_nLenMessOut.If the length of x_sMessageIn is greater than
  //  x_nLenMessOut it will be truncated.
  //  如果x_sMessageIn的消息长度是少于x_nLenMessOut的，增加空格。
  //  如果x_sMessageIn的消息长度是大于x_nLenMessOut的，将会被截断。
  //Input parameters
  //  string x_sMessageIn :
  //    role : Message that you want to display
  //    作用：你想去显示的消息
  //  num x_nLenMessOut :
  //    role : Length of the message out
  //    作用：输出消息的长度
  //Output parameters
  //  string x_sMessageOut :
  //    role : Message with spaces after or truncated if the length
  //          x_sMessageIn is greater than x_nLenMessOut
  //    作用：如果长度x_sMessageIn大于x_nLenMessOut，消息使用空格或被截断
  //Example
  //  call strFill("hello",20,l_sMessOut)
  //
  //History
  //  Creation : 28-04-08 - f.Rob
  //Header end
  //-----------------------------------------------------------------------
  //Look for asian message
  if getDisplayLen(x_sMessageIn)<x_nLenMessOut
    //Insert some spaces 插入一些空格
    l_sEmpty="                                        "
    x_sMessageOut=x_sMessageIn
    //Length of the spaces to add  增加空格的长度
    l_nLen=(x_nLenMessOut-getDisplayLen(x_sMessageIn))
    call midPos(l_sEmpty,l_nLen,0,x_sMessageIn)
    x_sMessageOut=x_sMessageOut+x_sMessageIn
  else
    if getDisplayLen(x_sMessageIn)>x_nLenMessOut
      //Divide the string  分割字符串
      call midPos(x_sMessageIn,x_nLenMessOut,0,x_sMessageOut)
    else
      //They are the same
      x_sMessageOut=x_sMessageIn
    endIf
  endIf
end

--- strFillChr.pgx ---
public program strFillChr(string x_sIn, string& x_sOut[], string x_sChar)
  local num l_nIndex
begin
  //-----------------------------------------------------------------------
  //Header begin
  //Description of program
  //  To fill the string with custom characters.
  //  Usually using for a cryptage.
  //  用一般字符来填充字符串，通常是用加密的方法。
  //Input parameters
  //  string x_sIn :
  //    role : string that you want modified
  //    作用：你想去修改的字符串
  //  string x_sChar :
  //    role : characters that you want replaced.
  //    作用：你想去替代的字符
  //Output parameters
  //  string x_sOut :
  //    role : string modified
  //   作用:修改的字符串
  //Example
  //   password cryptage
  //   call strFillChr(lPassword,lView,"*")
  //
  //History
  //  Creation : 28-04-08 - f.Rob
  //Header end
  //-----------------------------------------------------------------------
  x_sOut=""
  if getDisplayLen(x_sIn)>0
    for l_nIndex=0 to (getDisplayLen(x_sIn)-1)
      x_sOut=x_sOut+x_sChar
    endFor
  endIf
end

--- stringCopy.pgx ---
public program stringCopy(string& x_sCopy[], string& x_sPaste[])
// Copy all the value from the x_sCopy to x_sPaste
  local num i
  local num l_nSize
begin
  //-----------------------------------------------------------------------
  //Header begin
  //Description of program
  //  Copy all the values from the first parameter to the second one.
  //  从第一个参数中复制所有的值到第二个参数中
  //  You can copy an array of string.
  //  你可以复制一个字符串数组。
  //Input parameters
  //  string x_sCopy :
  //    role : string that you want to copy
  //    作用：你想去复制的字符串
  //  string x_sPaste :
  //    role : string paste
  //    作用：粘贴的字符串
  //Example
  //  call stringCopy("Robotics",sMessage)
  //
  //History
  //  Creation : 28-04-08 - f.Rob
  //Header end
  //-----------------------------------------------------------------------
  //Redim the Paste String ARRAY
  //Get the length of x_sPaste 得到x_sPaste的长度
  l_nSize=size(x_sPaste)
  if size(x_sCopy)>l_nSize
    //The length of x_sPaste is less than the length of x_sCopy  x_sPaste的长度是少于x_sCopy的长度的
    for i=l_nSize to (size(x_sCopy)-1)
      //Insert elements in the array x_sPaste at the 0 index 插入元素到数组x_sPaste到0索引的位置
      insert(x_sPaste[0])
    endFor
  else
    if size(x_sCopy)<size(x_sPaste)
      //The length of x_sCopy  is less than the length of x_sPaste
      for i=size(x_sCopy) to l_nSize-1
        //Destroy elements of the array x_sPaste at length of x_sCopy index
        delete(x_sPaste[0])
      endFor
    endIf
  endIf
  //Copy all the field
  for i=0 to (size(x_sCopy)-1)
    x_sPaste[i]=x_sCopy[i]
  endFor
end

--- stringToArray.pgx ---
public program stringToArray(string x_sString, string& x_sArray[])
// copy one String into an ARRAY of String
  local num i
  local num l_nItem
  local string l_sChar
  local string l_sEmpty
begin
  //-----------------------------------------------------------------------
  //Header begin
  //Description of program
  //  Copy one string into an array of string.  复制一个字符串到字符串数组
  //  Divide the string and add a box in the array when a specific  当找到一个特定的字符后，分割字符串，增加一个窗口到数组里。
  //  character was find.
  //  If the program find "^" in the string the char will be use to divide
  //  the items otherwise the char "," will be used.
  //  如果程序找到"^" 在字符串中，这个字符将被用来划分条目，否则字符","将被使用。
  //Input parameters
  //  string x_sString :
  //    role : string that you want to copy
  //    作用：你想要去复制的字符串
  //Output parameters
  //  string x_sArray :
  //    role : Array of string
  //    作用：字符串数组
  //Example
  //  call stringToArray("Stäubli,Robotics",sArray)
  //
  //History
  //  Creation : 28-04-08 - f.Rob
  //  Modified : 08-08-11 - J.Cook     Changed $setTextMode to setTextMode
  //                                   And replaced literals ("", 0) with local variables
  //                                   when passing parameters by reference
  //Header end
  //-----------------------------------------------------------------------
  //Defines the char used to divide the items 定义去分割条目的字符
  l_sEmpty = ""
  if find(x_sString,"^")==-1
    l_sChar=","
  else
    l_sChar="^"
  endIf
  //Init the x_sArray  初始化x_sArray
  call stringCopy(l_sEmpty,x_sArray)
  l_nItem=0
  do
    //Increase the ARRAY SIZE 增加数组的大小
    if l_nItem>0
      insert(x_sArray[l_nItem])
    endIf
    i=find(x_sString,l_sChar)
    //Look if was found 观察是否被找到
    if i!=-1
      //PUT INSIDE THE ARRAY THE STRING
      x_sArray[l_nItem]=left(x_sString,i)
      x_sString=delete(x_sString,i+1,0)
    else
      //Look if is empty or not 观察是否为空
      if len(x_sString)>0
        x_sArray[l_nItem]=(x_sString)
      endIf
    endIf
    l_nItem=l_nItem+1
  until i==-1
end

--- strlength.pgx ---
program strlength(string& x_sMessage[], num x_nLength)
  local string lStrEmpty
  local string l_sTemp
begin
  lStrEmpty="                                        "
  // Look for asian message
  if getDisplayLen(x_sMessage)>x_nLength
    // Need to divide the message 需要去分割消息
    if getDisplayLen(x_sMessage)==len(x_sMessage)
      if mid(x_sMessage,1,x_nLength)!=" "
        // European message
        x_sMessage=mid(x_sMessage,x_nLength-1,0)
        x_sMessage=x_sMessage+"."
      else
        // Found and empty space
        x_sMessage=mid(x_sMessage,x_nLength,0)
      endIf
    else
      // Asian one
      call midPos(x_sMessage,x_nLength,0,x_sMessage)
    endIf
  else
    if getDisplayLen(x_sMessage)<x_nLength
      // European
      if getDisplayLen(x_sMessage)==len(x_sMessage)
        x_sMessage=x_sMessage+mid(lStrEmpty,x_nLength-getDisplayLen(x_sMessage),0)
      else
        // Asian
        call midPos(lStrEmpty,x_nLength-getDisplayLen(x_sMessage),0,l_sTemp)
        x_sMessage=x_sMessage+l_sTemp
      endIf
    else
      // They are the same
    endIf
  endIf
end

--- test.pgx ---
program test(screen& x_scr)
  local num l_nItem
  local string sold[4]
begin
  call changeValue(x_scr,l_nItem,0,4,5,5,sTab)
end

